// TIA Portal V19 export
FUNCTION_BLOCK "A02_HMI_FB"   // FB175, LAD
TITLE = HMI Managment
AUTHOR : Piemme
FAMILY : System
// stored: MemoryReserve 100, SetENOAutomatically false
   VAR
      MB2_Decoder { ExternalAccessible := 'False'; ExternalVisible := 'False'; ExternalWritable := 'False'} : "ButtonsHMIDecoder";
   END_VAR
   VAR_TEMP
      i : Int;
      tempIdxMove : Int;
      tempIdxPos : Int;
      tempIdxVert : Int;
      tempIdxHoriz : Int;
   END_VAR
   VAR CONSTANT
      "2001_HU_AREA02" : Int := 2001;
      "2011_PIT_TABLE1" : Int := 2011;
      "2021_ROLLFORMER_MOVE" : Int := 2021;
      "2022_ROLLFORMER_LUBR_1" : Int := 2022;
      "2023_ROLLFORMER_LUBR_2" : Int := 2023;
      "2024_ROLLFORMER_LUBR_3" : Int := 2024;
      "2031_MWFAKCALC_PUSHAX" : Int := 2031;
      "2032_MWFAKCALC_GRIPPER" : Int := 2032;
      "2041_FLYINGCARRIAGE_MOVE" : Int := 2041;
      "2042_FLYINGCARRIAGE_POS" : Int := 2042;
      "2043_FLYINGCARRIAGE_ZERO" : Int := 2043;
      "2044_FLYINGCARRIAGE_LUBR" : Int := 2044;
      "2051_FINALCUT_LOCKING" : Int := 2051;
      "2052_FINALCUT_CUTHEAD" : Int := 2052;
      "2053_FINALCUT_DRAWHEAD" : Int := 2053;
      "2054_FINALCUT_MARKHEAD" : Int := 2054;
      "2055_FINALCUT_LUBR" : Int := 2055;
      "2061_ACCROLLCONVEYOR_COMBO_MOVE" : Int := 2061;
      "2062_ACCROLLCONVEYOR_PUSHER_COMBO_VERT" : Int := 2062;
      "2063_ACCROLLCONVEYOR_PUSHER_COMBO_HORIZ" : Int := 2063;
      "2071_ACCROLLCONVEYOR_ROLL1" : Int := 2071;
      "2072_ACCROLLCONVEYOR_ROLL2" : Int := 2072;
      "2073_ACCROLLCONVEYOR_ROLL3" : Int := 2073;
      "2081_ACCROLLCONVEYOR_PUSHER_VERT_1" : Int := 2081;
      "2082_ACCROLLCONVEYOR_PUSHER_VERT_2" : Int := 2082;
      "2083_ACCROLLCONVEYOR_PUSHER_VERT_3" : Int := 2083;
      "2084_ACCROLLCONVEYOR_PUSHER_VERT_4" : Int := 2084;
      "2085_ACCROLLCONVEYOR_PUSHER_VERT_5" : Int := 2085;
      "2086_ACCROLLCONVEYOR_PUSHER_VERT_6" : Int := 2086;
      "2091_ACCROLLCONVEYOR_PUSHER_HORIZ_1" : Int := 2091;
      "2092_ACCROLLCONVEYOR_PUSHER_HORIZ_2" : Int := 2092;
      "2093_ACCROLLCONVEYOR_PUSHER_HORIZ_3" : Int := 2093;
      "2094_ACCROLLCONVEYOR_PUSHER_HORIZ_4" : Int := 2094;
      "2095_ACCROLLCONVEYOR_PUSHER_HORIZ_5" : Int := 2095;
      "2096_ACCROLLCONVEYOR_PUSHER_HORIZ_6" : Int := 2096;
      "2100_MODULO1_OP_MOVE" : Int := 2100;
      "2101_MODULO1_OP_POS" : Int := 2101;
      "2102_MODULO1_MOT_MOVE" : Int := 2102;
      "2103_MODULO1_MOT_POS" : Int := 2103;
      "2104_MODULO2_OP_MOVE" : Int := 2104;
      "2105_MODULO2_OP_POS" : Int := 2105;
      "2106_MODULO2_MOT_MOVE" : Int := 2106;
      "2107_MODULO2_MOT_POS" : Int := 2107;
      "2108_MODULO3_OP_MOVE" : Int := 2108;
      "2109_MODULO3_OP_POS" : Int := 2109;
      "2110_MODULO3_MOT_MOVE" : Int := 2110;
      "2111_MODULO3_MOT_POS" : Int := 2111;
      "2112_PASSAGGIO2_OP_MOVE" : Int := 2112;
      "2113_PASSAGGIO2_OP_POS" : Int := 2113;
      "2114_PASSAGGIO2_MOT_MOVE" : Int := 2114;
      "2115_PASSAGGIO2_MOT_POS" : Int := 2115;
      "2116_PASSAGGIO14_OP_MOVE" : Int := 2116;
      "2117_PASSAGGIO14_OP_POS" : Int := 2117;
      "2118_PASSAGGIO14_MOT_MOVE" : Int := 2118;
      "2119_PASSAGGIO14_MOT_POS" : Int := 2119;
      "2120_PASSAGGIO17_OP_MOVE" : Int := 2120;
      "2121_PASSAGGIO17_OP_POS" : Int := 2121;
      "2122_PASSAGGIO17_MOT_MOVE" : Int := 2122;
      "2123_PASSAGGIO17_MOT_POS" : Int := 2123;
      "2124_PASSAGGIO18_OP_MOVE" : Int := 2124;
      "2125_PASSAGGIO18_OP_POS" : Int := 2125;
      "2126_PASSAGGIO18_MOT_MOVE" : Int := 2126;
      "2127_PASSAGGIO18_MOT_POS" : Int := 2127;
      "2280_PASSAGGIO2_COMBO_MOVE" : Int := 2280;
      "2281_PASSAGGIO2_COMBO_POS" : Int := 2281;
      "2282_PASSAGGIO14_COMBO_MOVE" : Int := 2282;
      "2283_PASSAGGIO14_COMBO_POS" : Int := 2283;
      "2284_PASSAGGIO17_COMBO_MOVE" : Int := 2284;
      "2285_PASSAGGIO17_COMBO_POS" : Int := 2285;
      "2286_PASSAGGIO18_COMBO_MOVE" : Int := 2286;
      "2287_PASSAGGIO18_COMBO_POS" : Int := 2287;
   END_VAR
   VAR_TEMP   // added for the SCL form of the ladder/FBD networks
      _w1 : Bool;
   END_VAR
BEGIN

REGION Network 2: <<< MB2 MANUALS OPERATIONS >>>
END_REGION

REGION Network 3 (SCL): Reset Op
   #MB2_Decoder.OpEnabled := FALSE;
   #MB2_Decoder.OpRunning := FALSE;
   #MB2_Decoder.OpDone := FALSE;
END_REGION

REGION Network 4: MB2 Code 2001 - Area 02 HU
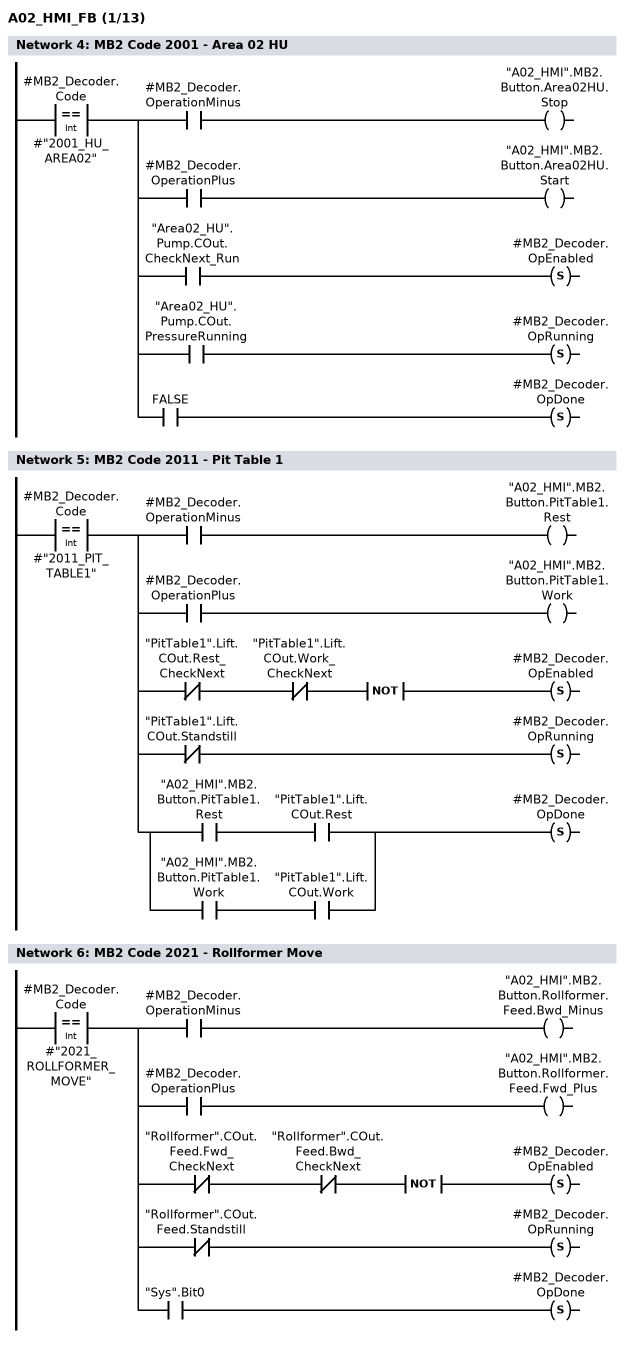
   RUNG wire#powerrail
      { S7_Templates := "SrcType := Int" } EQ_Contact(in1 := #MB2_Decoder.Code, in2 := #"2001_HU_AREA02")
      wire#w1
      Contact( #MB2_Decoder.OperationMinus )
      Coil( "A02_HMI".MB2.Button.Area02HU.Stop )
   END_RUNG
   RUNG wire#w1
      Contact( #MB2_Decoder.OperationPlus )
      Coil( "A02_HMI".MB2.Button.Area02HU.Start )
   END_RUNG
   RUNG wire#w1
      Contact( "Area02_HU".Pump.COut.CheckNext_Run )
      S_Coil( #MB2_Decoder.OpEnabled )
   END_RUNG
   RUNG wire#w1
      Contact( "Area02_HU".Pump.COut.PressureRunning )
      S_Coil( #MB2_Decoder.OpRunning )
   END_RUNG
   RUNG wire#w1
      Contact( FALSE )
      S_Coil( #MB2_Decoder.OpDone )
   END_RUNG
   // the same network as SCL:
   #_w1 := #MB2_Decoder.Code = #"2001_HU_AREA02";
   "A02_HMI".MB2.Button.Area02HU.Stop := #_w1 AND #MB2_Decoder.OperationMinus;
   "A02_HMI".MB2.Button.Area02HU.Start := #_w1 AND #MB2_Decoder.OperationPlus;
   IF #_w1 AND "Area02_HU".Pump.COut.CheckNext_Run THEN #MB2_Decoder.OpEnabled := TRUE; END_IF;
   IF #_w1 AND "Area02_HU".Pump.COut.PressureRunning THEN #MB2_Decoder.OpRunning := TRUE; END_IF;
   IF #_w1 AND FALSE THEN #MB2_Decoder.OpDone := TRUE; END_IF;
END_REGION

REGION Network 5: MB2 Code 2011 - Pit Table 1
   RUNG wire#powerrail
      { S7_Templates := "SrcType := Int" } EQ_Contact(in1 := #MB2_Decoder.Code, in2 := #"2011_PIT_TABLE1")
      wire#w1
      Contact( #MB2_Decoder.OperationMinus )
      Coil( "A02_HMI".MB2.Button.PitTable1.Rest )
   END_RUNG
   RUNG wire#w1
      Contact( #MB2_Decoder.OperationPlus )
      Coil( "A02_HMI".MB2.Button.PitTable1.Work )
   END_RUNG
   RUNG wire#w1
      I_Contact( "PitTable1".Lift.COut.Rest_CheckNext )
      I_Contact( "PitTable1".Lift.COut.Work_CheckNext )
      Not()
      S_Coil( #MB2_Decoder.OpEnabled )
   END_RUNG
   RUNG wire#w1
      I_Contact( "PitTable1".Lift.COut.Standstill )
      S_Coil( #MB2_Decoder.OpRunning )
   END_RUNG
   RUNG wire#w1
      Contact( "A02_HMI".MB2.Button.PitTable1.Rest )
      Contact( "PitTable1".Lift.COut.Rest )
      wire#w2
      S_Coil( #MB2_Decoder.OpDone )
   END_RUNG
   RUNG wire#w1
      Contact( "A02_HMI".MB2.Button.PitTable1.Work )
      Contact( "PitTable1".Lift.COut.Work )
   END_RUNG wire#w2
   // the same network as SCL:
   #_w1 := #MB2_Decoder.Code = #"2011_PIT_TABLE1";
   "A02_HMI".MB2.Button.PitTable1.Rest := #_w1 AND #MB2_Decoder.OperationMinus;
   "A02_HMI".MB2.Button.PitTable1.Work := #_w1 AND #MB2_Decoder.OperationPlus;
   IF NOT (#_w1 AND NOT "PitTable1".Lift.COut.Rest_CheckNext AND NOT "PitTable1".Lift.COut.Work_CheckNext) THEN
       #MB2_Decoder.OpEnabled := TRUE;
   END_IF;
   IF #_w1 AND NOT "PitTable1".Lift.COut.Standstill THEN #MB2_Decoder.OpRunning := TRUE; END_IF;
   IF #_w1 AND (("A02_HMI".MB2.Button.PitTable1.Rest AND "PitTable1".Lift.COut.Rest) OR ("A02_HMI".MB2.Button.PitTable1.Work AND "PitTable1".Lift.COut.Work)) THEN
       #MB2_Decoder.OpDone := TRUE;
   END_IF;
END_REGION

REGION Network 6: MB2 Code 2021 - Rollformer Move
   RUNG wire#powerrail
      { S7_Templates := "SrcType := Int" } EQ_Contact(in1 := #MB2_Decoder.Code, in2 := #"2021_ROLLFORMER_MOVE")
      wire#w1
      Contact( #MB2_Decoder.OperationMinus )
      Coil( "A02_HMI".MB2.Button.Rollformer.Feed.Bwd_Minus )
   END_RUNG
   RUNG wire#w1
      Contact( #MB2_Decoder.OperationPlus )
      Coil( "A02_HMI".MB2.Button.Rollformer.Feed.Fwd_Plus )
   END_RUNG
   RUNG wire#w1
      I_Contact( "Rollformer".COut.Feed.Fwd_CheckNext )
      I_Contact( "Rollformer".COut.Feed.Bwd_CheckNext )
      Not()
      S_Coil( #MB2_Decoder.OpEnabled )
   END_RUNG
   RUNG wire#w1
      I_Contact( "Rollformer".COut.Feed.Standstill )
      S_Coil( #MB2_Decoder.OpRunning )
   END_RUNG
   RUNG wire#w1
      Contact( "Sys".Bit0 )
      S_Coil( #MB2_Decoder.OpDone )
   END_RUNG
   // the same network as SCL:
   #_w1 := #MB2_Decoder.Code = #"2021_ROLLFORMER_MOVE";
   "A02_HMI".MB2.Button.Rollformer.Feed.Bwd_Minus := #_w1 AND #MB2_Decoder.OperationMinus;
   "A02_HMI".MB2.Button.Rollformer.Feed.Fwd_Plus := #_w1 AND #MB2_Decoder.OperationPlus;
   IF NOT (#_w1 AND NOT "Rollformer".COut.Feed.Fwd_CheckNext AND NOT "Rollformer".COut.Feed.Bwd_CheckNext) THEN
       #MB2_Decoder.OpEnabled := TRUE;
   END_IF;
   IF #_w1 AND NOT "Rollformer".COut.Feed.Standstill THEN #MB2_Decoder.OpRunning := TRUE; END_IF;
   IF #_w1 AND "Sys".Bit0 THEN #MB2_Decoder.OpDone := TRUE; END_IF;
END_REGION

REGION Network 7: MB2 Code 2022 - Rollformer Lubr 1
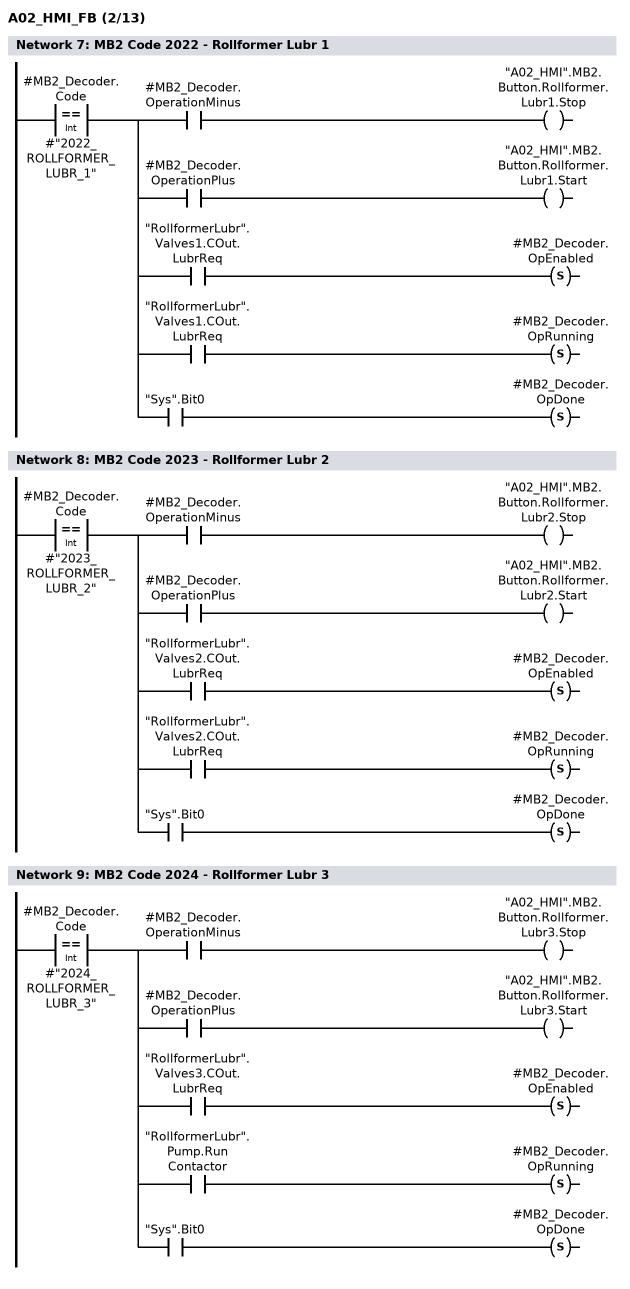
   RUNG wire#powerrail
      { S7_Templates := "SrcType := Int" } EQ_Contact(in1 := #MB2_Decoder.Code, in2 := #"2022_ROLLFORMER_LUBR_1")
      wire#w1
      Contact( #MB2_Decoder.OperationMinus )
      Coil( "A02_HMI".MB2.Button.Rollformer.Lubr1.Stop )
   END_RUNG
   RUNG wire#w1
      Contact( #MB2_Decoder.OperationPlus )
      Coil( "A02_HMI".MB2.Button.Rollformer.Lubr1.Start )
   END_RUNG
   RUNG wire#w1
      Contact( "RollformerLubr".Valves1.COut.LubrReq )
      S_Coil( #MB2_Decoder.OpEnabled )
   END_RUNG
   RUNG wire#w1
      Contact( "RollformerLubr".Valves1.COut.LubrReq )
      S_Coil( #MB2_Decoder.OpRunning )
   END_RUNG
   RUNG wire#w1
      Contact( "Sys".Bit0 )
      S_Coil( #MB2_Decoder.OpDone )
   END_RUNG
   // the same network as SCL:
   #_w1 := #MB2_Decoder.Code = #"2022_ROLLFORMER_LUBR_1";
   "A02_HMI".MB2.Button.Rollformer.Lubr1.Stop := #_w1 AND #MB2_Decoder.OperationMinus;
   "A02_HMI".MB2.Button.Rollformer.Lubr1.Start := #_w1 AND #MB2_Decoder.OperationPlus;
   IF #_w1 AND "RollformerLubr".Valves1.COut.LubrReq THEN
       #MB2_Decoder.OpEnabled := TRUE;
       #MB2_Decoder.OpRunning := TRUE;
   END_IF;
   IF #_w1 AND "Sys".Bit0 THEN #MB2_Decoder.OpDone := TRUE; END_IF;
END_REGION

REGION Network 8: MB2 Code 2023 - Rollformer Lubr 2
   RUNG wire#powerrail
      { S7_Templates := "SrcType := Int" } EQ_Contact(in1 := #MB2_Decoder.Code, in2 := #"2023_ROLLFORMER_LUBR_2")
      wire#w1
      Contact( #MB2_Decoder.OperationMinus )
      Coil( "A02_HMI".MB2.Button.Rollformer.Lubr2.Stop )
   END_RUNG
   RUNG wire#w1
      Contact( #MB2_Decoder.OperationPlus )
      Coil( "A02_HMI".MB2.Button.Rollformer.Lubr2.Start )
   END_RUNG
   RUNG wire#w1
      Contact( "RollformerLubr".Valves2.COut.LubrReq )
      S_Coil( #MB2_Decoder.OpEnabled )
   END_RUNG
   RUNG wire#w1
      Contact( "RollformerLubr".Valves2.COut.LubrReq )
      S_Coil( #MB2_Decoder.OpRunning )
   END_RUNG
   RUNG wire#w1
      Contact( "Sys".Bit0 )
      S_Coil( #MB2_Decoder.OpDone )
   END_RUNG
   // the same network as SCL:
   #_w1 := #MB2_Decoder.Code = #"2023_ROLLFORMER_LUBR_2";
   "A02_HMI".MB2.Button.Rollformer.Lubr2.Stop := #_w1 AND #MB2_Decoder.OperationMinus;
   "A02_HMI".MB2.Button.Rollformer.Lubr2.Start := #_w1 AND #MB2_Decoder.OperationPlus;
   IF #_w1 AND "RollformerLubr".Valves2.COut.LubrReq THEN
       #MB2_Decoder.OpEnabled := TRUE;
       #MB2_Decoder.OpRunning := TRUE;
   END_IF;
   IF #_w1 AND "Sys".Bit0 THEN #MB2_Decoder.OpDone := TRUE; END_IF;
END_REGION

REGION Network 9: MB2 Code 2024 - Rollformer Lubr 3
   RUNG wire#powerrail
      { S7_Templates := "SrcType := Int" } EQ_Contact(in1 := #MB2_Decoder.Code, in2 := #"2024_ROLLFORMER_LUBR_3")
      wire#w1
      Contact( #MB2_Decoder.OperationMinus )
      Coil( "A02_HMI".MB2.Button.Rollformer.Lubr3.Stop )
   END_RUNG
   RUNG wire#w1
      Contact( #MB2_Decoder.OperationPlus )
      Coil( "A02_HMI".MB2.Button.Rollformer.Lubr3.Start )
   END_RUNG
   RUNG wire#w1
      Contact( "RollformerLubr".Valves3.COut.LubrReq )
      S_Coil( #MB2_Decoder.OpEnabled )
   END_RUNG
   RUNG wire#w1
      Contact( "RollformerLubr".Pump.RunContactor )
      S_Coil( #MB2_Decoder.OpRunning )
   END_RUNG
   RUNG wire#w1
      Contact( "Sys".Bit0 )
      S_Coil( #MB2_Decoder.OpDone )
   END_RUNG
   // the same network as SCL:
   #_w1 := #MB2_Decoder.Code = #"2024_ROLLFORMER_LUBR_3";
   "A02_HMI".MB2.Button.Rollformer.Lubr3.Stop := #_w1 AND #MB2_Decoder.OperationMinus;
   "A02_HMI".MB2.Button.Rollformer.Lubr3.Start := #_w1 AND #MB2_Decoder.OperationPlus;
   IF #_w1 AND "RollformerLubr".Valves3.COut.LubrReq THEN #MB2_Decoder.OpEnabled := TRUE; END_IF;
   IF #_w1 AND "RollformerLubr".Pump.RunContactor THEN #MB2_Decoder.OpRunning := TRUE; END_IF;
   IF #_w1 AND "Sys".Bit0 THEN #MB2_Decoder.OpDone := TRUE; END_IF;
END_REGION

REGION Network 10: MB2 Code 2031 - MwFakCalc push ax
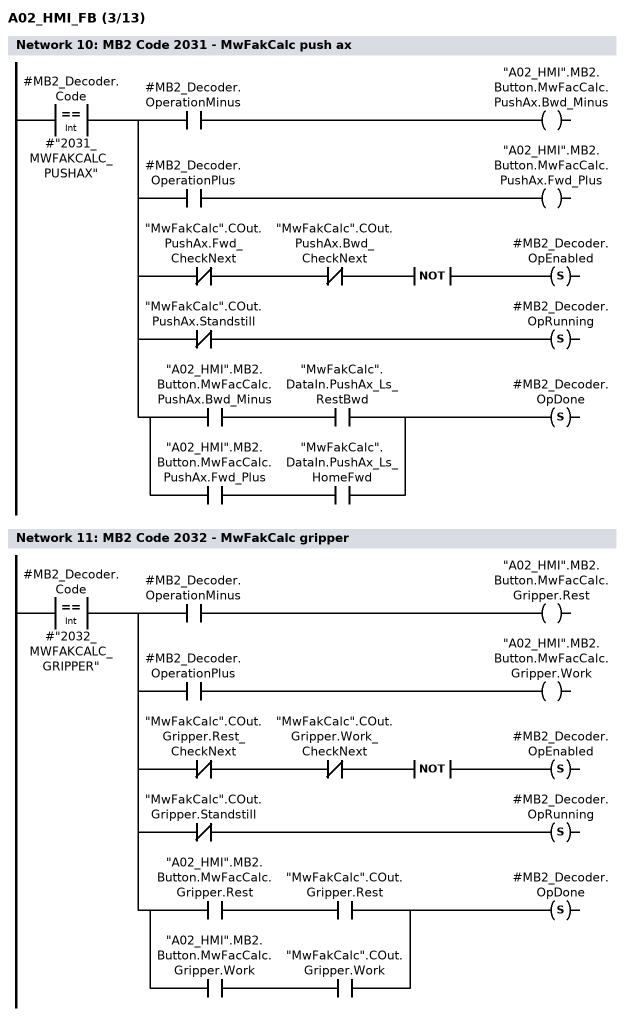
   RUNG wire#powerrail
      { S7_Templates := "SrcType := Int" } EQ_Contact(in1 := #MB2_Decoder.Code, in2 := #"2031_MWFAKCALC_PUSHAX")
      wire#w1
      Contact( #MB2_Decoder.OperationMinus )
      Coil( "A02_HMI".MB2.Button.MwFacCalc.PushAx.Bwd_Minus )
   END_RUNG
   RUNG wire#w1
      Contact( #MB2_Decoder.OperationPlus )
      Coil( "A02_HMI".MB2.Button.MwFacCalc.PushAx.Fwd_Plus )
   END_RUNG
   RUNG wire#w1
      I_Contact( "MwFakCalc".COut.PushAx.Fwd_CheckNext )
      I_Contact( "MwFakCalc".COut.PushAx.Bwd_CheckNext )
      Not()
      S_Coil( #MB2_Decoder.OpEnabled )
   END_RUNG
   RUNG wire#w1
      I_Contact( "MwFakCalc".COut.PushAx.Standstill )
      S_Coil( #MB2_Decoder.OpRunning )
   END_RUNG
   RUNG wire#w1
      Contact( "A02_HMI".MB2.Button.MwFacCalc.PushAx.Bwd_Minus )
      Contact( "MwFakCalc".DataIn.PushAx_Ls_RestBwd )
      wire#w2
      S_Coil( #MB2_Decoder.OpDone )
   END_RUNG
   RUNG wire#w1
      Contact( "A02_HMI".MB2.Button.MwFacCalc.PushAx.Fwd_Plus )
      Contact( "MwFakCalc".DataIn.PushAx_Ls_HomeFwd )
   END_RUNG wire#w2
   // the same network as SCL:
   #_w1 := #MB2_Decoder.Code = #"2031_MWFAKCALC_PUSHAX";
   "A02_HMI".MB2.Button.MwFacCalc.PushAx.Bwd_Minus := #_w1 AND #MB2_Decoder.OperationMinus;
   "A02_HMI".MB2.Button.MwFacCalc.PushAx.Fwd_Plus := #_w1 AND #MB2_Decoder.OperationPlus;
   IF NOT (#_w1 AND NOT "MwFakCalc".COut.PushAx.Fwd_CheckNext AND NOT "MwFakCalc".COut.PushAx.Bwd_CheckNext) THEN
       #MB2_Decoder.OpEnabled := TRUE;
   END_IF;
   IF #_w1 AND NOT "MwFakCalc".COut.PushAx.Standstill THEN #MB2_Decoder.OpRunning := TRUE; END_IF;
   IF #_w1 AND (("A02_HMI".MB2.Button.MwFacCalc.PushAx.Bwd_Minus AND "MwFakCalc".DataIn.PushAx_Ls_RestBwd) OR ("A02_HMI".MB2.Button.MwFacCalc.PushAx.Fwd_Plus AND "MwFakCalc".DataIn.PushAx_Ls_HomeFwd)) THEN
       #MB2_Decoder.OpDone := TRUE;
   END_IF;
END_REGION

REGION Network 11: MB2 Code 2032 - MwFakCalc gripper
   RUNG wire#powerrail
      { S7_Templates := "SrcType := Int" } EQ_Contact(in1 := #MB2_Decoder.Code, in2 := #"2032_MWFAKCALC_GRIPPER")
      wire#w1
      Contact( #MB2_Decoder.OperationMinus )
      Coil( "A02_HMI".MB2.Button.MwFacCalc.Gripper.Rest )
   END_RUNG
   RUNG wire#w1
      Contact( #MB2_Decoder.OperationPlus )
      Coil( "A02_HMI".MB2.Button.MwFacCalc.Gripper.Work )
   END_RUNG
   RUNG wire#w1
      I_Contact( "MwFakCalc".COut.Gripper.Rest_CheckNext )
      I_Contact( "MwFakCalc".COut.Gripper.Work_CheckNext )
      Not()
      S_Coil( #MB2_Decoder.OpEnabled )
   END_RUNG
   RUNG wire#w1
      I_Contact( "MwFakCalc".COut.Gripper.Standstill )
      S_Coil( #MB2_Decoder.OpRunning )
   END_RUNG
   RUNG wire#w1
      Contact( "A02_HMI".MB2.Button.MwFacCalc.Gripper.Rest )
      Contact( "MwFakCalc".COut.Gripper.Rest )
      wire#w2
      S_Coil( #MB2_Decoder.OpDone )
   END_RUNG
   RUNG wire#w1
      Contact( "A02_HMI".MB2.Button.MwFacCalc.Gripper.Work )
      Contact( "MwFakCalc".COut.Gripper.Work )
   END_RUNG wire#w2
   // the same network as SCL:
   #_w1 := #MB2_Decoder.Code = #"2032_MWFAKCALC_GRIPPER";
   "A02_HMI".MB2.Button.MwFacCalc.Gripper.Rest := #_w1 AND #MB2_Decoder.OperationMinus;
   "A02_HMI".MB2.Button.MwFacCalc.Gripper.Work := #_w1 AND #MB2_Decoder.OperationPlus;
   IF NOT (#_w1 AND NOT "MwFakCalc".COut.Gripper.Rest_CheckNext AND NOT "MwFakCalc".COut.Gripper.Work_CheckNext) THEN
       #MB2_Decoder.OpEnabled := TRUE;
   END_IF;
   IF #_w1 AND NOT "MwFakCalc".COut.Gripper.Standstill THEN #MB2_Decoder.OpRunning := TRUE; END_IF;
   IF #_w1 AND (("A02_HMI".MB2.Button.MwFacCalc.Gripper.Rest AND "MwFakCalc".COut.Gripper.Rest) OR ("A02_HMI".MB2.Button.MwFacCalc.Gripper.Work AND "MwFakCalc".COut.Gripper.Work)) THEN
       #MB2_Decoder.OpDone := TRUE;
   END_IF;
END_REGION

REGION Network 12: MB2 Code 2041 - Flying carriage move
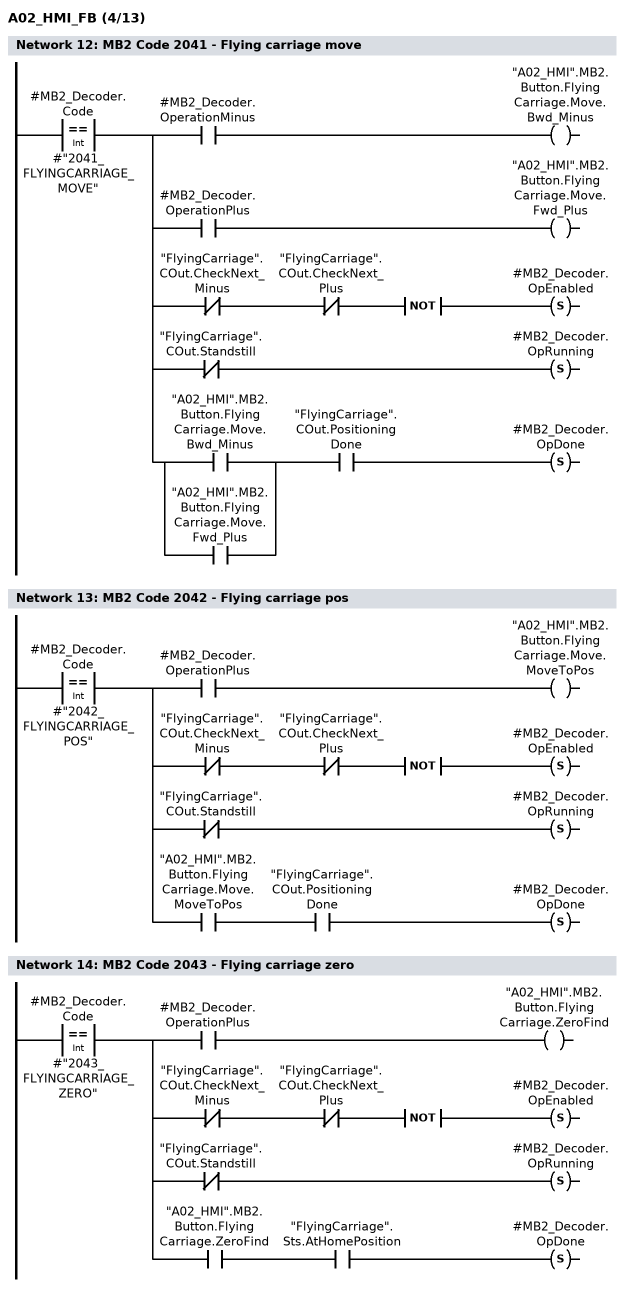
   RUNG wire#powerrail
      { S7_Templates := "SrcType := Int" } EQ_Contact(in1 := #MB2_Decoder.Code, in2 := #"2041_FLYINGCARRIAGE_MOVE")
      wire#w1
      Contact( #MB2_Decoder.OperationMinus )
      Coil( "A02_HMI".MB2.Button.FlyingCarriage.Move.Bwd_Minus )
   END_RUNG
   RUNG wire#w1
      Contact( #MB2_Decoder.OperationPlus )
      Coil( "A02_HMI".MB2.Button.FlyingCarriage.Move.Fwd_Plus )
   END_RUNG
   RUNG wire#w1
      I_Contact( "FlyingCarriage".COut.CheckNext_Minus )
      I_Contact( "FlyingCarriage".COut.CheckNext_Plus )
      Not()
      S_Coil( #MB2_Decoder.OpEnabled )
   END_RUNG
   RUNG wire#w1
      I_Contact( "FlyingCarriage".COut.Standstill )
      S_Coil( #MB2_Decoder.OpRunning )
   END_RUNG
   RUNG wire#w1
      Contact( "A02_HMI".MB2.Button.FlyingCarriage.Move.Bwd_Minus )
      wire#w2
      Contact( "FlyingCarriage".COut.PositioningDone )
      S_Coil( #MB2_Decoder.OpDone )
   END_RUNG
   RUNG wire#w1
      Contact( "A02_HMI".MB2.Button.FlyingCarriage.Move.Fwd_Plus )
   END_RUNG wire#w2
   // the same network as SCL:
   #_w1 := #MB2_Decoder.Code = #"2041_FLYINGCARRIAGE_MOVE";
   "A02_HMI".MB2.Button.FlyingCarriage.Move.Bwd_Minus := #_w1 AND #MB2_Decoder.OperationMinus;
   "A02_HMI".MB2.Button.FlyingCarriage.Move.Fwd_Plus := #_w1 AND #MB2_Decoder.OperationPlus;
   IF NOT (#_w1 AND NOT "FlyingCarriage".COut.CheckNext_Minus AND NOT "FlyingCarriage".COut.CheckNext_Plus) THEN
       #MB2_Decoder.OpEnabled := TRUE;
   END_IF;
   IF #_w1 AND NOT "FlyingCarriage".COut.Standstill THEN #MB2_Decoder.OpRunning := TRUE; END_IF;
   IF #_w1 AND ("A02_HMI".MB2.Button.FlyingCarriage.Move.Bwd_Minus OR "A02_HMI".MB2.Button.FlyingCarriage.Move.Fwd_Plus) AND "FlyingCarriage".COut.PositioningDone THEN
       #MB2_Decoder.OpDone := TRUE;
   END_IF;
END_REGION

REGION Network 13: MB2 Code 2042 - Flying carriage pos
   RUNG wire#powerrail
      { S7_Templates := "SrcType := Int" } EQ_Contact(in1 := #MB2_Decoder.Code, in2 := #"2042_FLYINGCARRIAGE_POS")
      wire#w1
      Contact( #MB2_Decoder.OperationPlus )
      Coil( "A02_HMI".MB2.Button.FlyingCarriage.Move.MoveToPos )
   END_RUNG
   RUNG wire#w1
      I_Contact( "FlyingCarriage".COut.CheckNext_Minus )
      I_Contact( "FlyingCarriage".COut.CheckNext_Plus )
      Not()
      S_Coil( #MB2_Decoder.OpEnabled )
   END_RUNG
   RUNG wire#w1
      I_Contact( "FlyingCarriage".COut.Standstill )
      S_Coil( #MB2_Decoder.OpRunning )
   END_RUNG
   RUNG wire#w1
      Contact( "A02_HMI".MB2.Button.FlyingCarriage.Move.MoveToPos )
      Contact( "FlyingCarriage".COut.PositioningDone )
      S_Coil( #MB2_Decoder.OpDone )
   END_RUNG
   // the same network as SCL:
   #_w1 := #MB2_Decoder.Code = #"2042_FLYINGCARRIAGE_POS";
   "A02_HMI".MB2.Button.FlyingCarriage.Move.MoveToPos := #_w1 AND #MB2_Decoder.OperationPlus;
   IF NOT (#_w1 AND NOT "FlyingCarriage".COut.CheckNext_Minus AND NOT "FlyingCarriage".COut.CheckNext_Plus) THEN
       #MB2_Decoder.OpEnabled := TRUE;
   END_IF;
   IF #_w1 AND NOT "FlyingCarriage".COut.Standstill THEN #MB2_Decoder.OpRunning := TRUE; END_IF;
   IF #_w1 AND "A02_HMI".MB2.Button.FlyingCarriage.Move.MoveToPos AND "FlyingCarriage".COut.PositioningDone THEN
       #MB2_Decoder.OpDone := TRUE;
   END_IF;
END_REGION

REGION Network 14: MB2 Code 2043 - Flying carriage zero
   RUNG wire#powerrail
      { S7_Templates := "SrcType := Int" } EQ_Contact(in1 := #MB2_Decoder.Code, in2 := #"2043_FLYINGCARRIAGE_ZERO")
      wire#w1
      Contact( #MB2_Decoder.OperationPlus )
      Coil( "A02_HMI".MB2.Button.FlyingCarriage.ZeroFind )
   END_RUNG
   RUNG wire#w1
      I_Contact( "FlyingCarriage".COut.CheckNext_Minus )
      I_Contact( "FlyingCarriage".COut.CheckNext_Plus )
      Not()
      S_Coil( #MB2_Decoder.OpEnabled )
   END_RUNG
   RUNG wire#w1
      I_Contact( "FlyingCarriage".COut.Standstill )
      S_Coil( #MB2_Decoder.OpRunning )
   END_RUNG
   RUNG wire#w1
      Contact( "A02_HMI".MB2.Button.FlyingCarriage.ZeroFind )
      Contact( "FlyingCarriage".Sts.AtHomePosition )
      S_Coil( #MB2_Decoder.OpDone )
   END_RUNG
   // the same network as SCL:
   #_w1 := #MB2_Decoder.Code = #"2043_FLYINGCARRIAGE_ZERO";
   "A02_HMI".MB2.Button.FlyingCarriage.ZeroFind := #_w1 AND #MB2_Decoder.OperationPlus;
   IF NOT (#_w1 AND NOT "FlyingCarriage".COut.CheckNext_Minus AND NOT "FlyingCarriage".COut.CheckNext_Plus) THEN
       #MB2_Decoder.OpEnabled := TRUE;
   END_IF;
   IF #_w1 AND NOT "FlyingCarriage".COut.Standstill THEN #MB2_Decoder.OpRunning := TRUE; END_IF;
   IF #_w1 AND "A02_HMI".MB2.Button.FlyingCarriage.ZeroFind AND "FlyingCarriage".Sts.AtHomePosition THEN
       #MB2_Decoder.OpDone := TRUE;
   END_IF;
END_REGION

REGION Network 15: MB2 Code 2044 - Flying carriage lubr
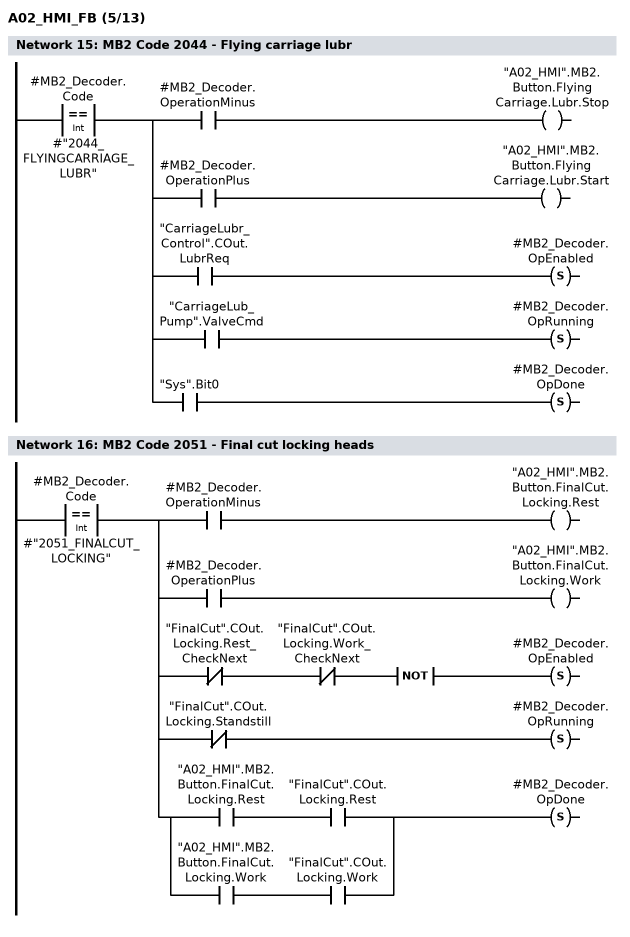
   RUNG wire#powerrail
      { S7_Templates := "SrcType := Int" } EQ_Contact(in1 := #MB2_Decoder.Code, in2 := #"2044_FLYINGCARRIAGE_LUBR")
      wire#w1
      Contact( #MB2_Decoder.OperationMinus )
      Coil( "A02_HMI".MB2.Button.FlyingCarriage.Lubr.Stop )
   END_RUNG
   RUNG wire#w1
      Contact( #MB2_Decoder.OperationPlus )
      Coil( "A02_HMI".MB2.Button.FlyingCarriage.Lubr.Start )
   END_RUNG
   RUNG wire#w1
      Contact( "CarriageLubr_Control".COut.LubrReq )
      S_Coil( #MB2_Decoder.OpEnabled )
   END_RUNG
   RUNG wire#w1
      Contact( "CarriageLub_Pump".ValveCmd )
      S_Coil( #MB2_Decoder.OpRunning )
   END_RUNG
   RUNG wire#w1
      Contact( "Sys".Bit0 )
      S_Coil( #MB2_Decoder.OpDone )
   END_RUNG
   // the same network as SCL:
   #_w1 := #MB2_Decoder.Code = #"2044_FLYINGCARRIAGE_LUBR";
   "A02_HMI".MB2.Button.FlyingCarriage.Lubr.Stop := #_w1 AND #MB2_Decoder.OperationMinus;
   "A02_HMI".MB2.Button.FlyingCarriage.Lubr.Start := #_w1 AND #MB2_Decoder.OperationPlus;
   IF #_w1 AND "CarriageLubr_Control".COut.LubrReq THEN #MB2_Decoder.OpEnabled := TRUE; END_IF;
   IF #_w1 AND "CarriageLub_Pump".ValveCmd THEN #MB2_Decoder.OpRunning := TRUE; END_IF;
   IF #_w1 AND "Sys".Bit0 THEN #MB2_Decoder.OpDone := TRUE; END_IF;
END_REGION

REGION Network 16: MB2 Code 2051 - Final cut locking heads
   RUNG wire#powerrail
      { S7_Templates := "SrcType := Int" } EQ_Contact(in1 := #MB2_Decoder.Code, in2 := #"2051_FINALCUT_LOCKING")
      wire#w1
      Contact( #MB2_Decoder.OperationMinus )
      Coil( "A02_HMI".MB2.Button.FinalCut.Locking.Rest )
   END_RUNG
   RUNG wire#w1
      Contact( #MB2_Decoder.OperationPlus )
      Coil( "A02_HMI".MB2.Button.FinalCut.Locking.Work )
   END_RUNG
   RUNG wire#w1
      I_Contact( "FinalCut".COut.Locking.Rest_CheckNext )
      I_Contact( "FinalCut".COut.Locking.Work_CheckNext )
      Not()
      S_Coil( #MB2_Decoder.OpEnabled )
   END_RUNG
   RUNG wire#w1
      I_Contact( "FinalCut".COut.Locking.Standstill )
      S_Coil( #MB2_Decoder.OpRunning )
   END_RUNG
   RUNG wire#w1
      Contact( "A02_HMI".MB2.Button.FinalCut.Locking.Rest )
      Contact( "FinalCut".COut.Locking.Rest )
      wire#w2
      S_Coil( #MB2_Decoder.OpDone )
   END_RUNG
   RUNG wire#w1
      Contact( "A02_HMI".MB2.Button.FinalCut.Locking.Work )
      Contact( "FinalCut".COut.Locking.Work )
   END_RUNG wire#w2
   // the same network as SCL:
   #_w1 := #MB2_Decoder.Code = #"2051_FINALCUT_LOCKING";
   "A02_HMI".MB2.Button.FinalCut.Locking.Rest := #_w1 AND #MB2_Decoder.OperationMinus;
   "A02_HMI".MB2.Button.FinalCut.Locking.Work := #_w1 AND #MB2_Decoder.OperationPlus;
   IF NOT (#_w1 AND NOT "FinalCut".COut.Locking.Rest_CheckNext AND NOT "FinalCut".COut.Locking.Work_CheckNext) THEN
       #MB2_Decoder.OpEnabled := TRUE;
   END_IF;
   IF #_w1 AND NOT "FinalCut".COut.Locking.Standstill THEN #MB2_Decoder.OpRunning := TRUE; END_IF;
   IF #_w1 AND (("A02_HMI".MB2.Button.FinalCut.Locking.Rest AND "FinalCut".COut.Locking.Rest) OR ("A02_HMI".MB2.Button.FinalCut.Locking.Work AND "FinalCut".COut.Locking.Work)) THEN
       #MB2_Decoder.OpDone := TRUE;
   END_IF;
END_REGION

REGION Network 17: MB2 Code 2052 - Final cut cut head
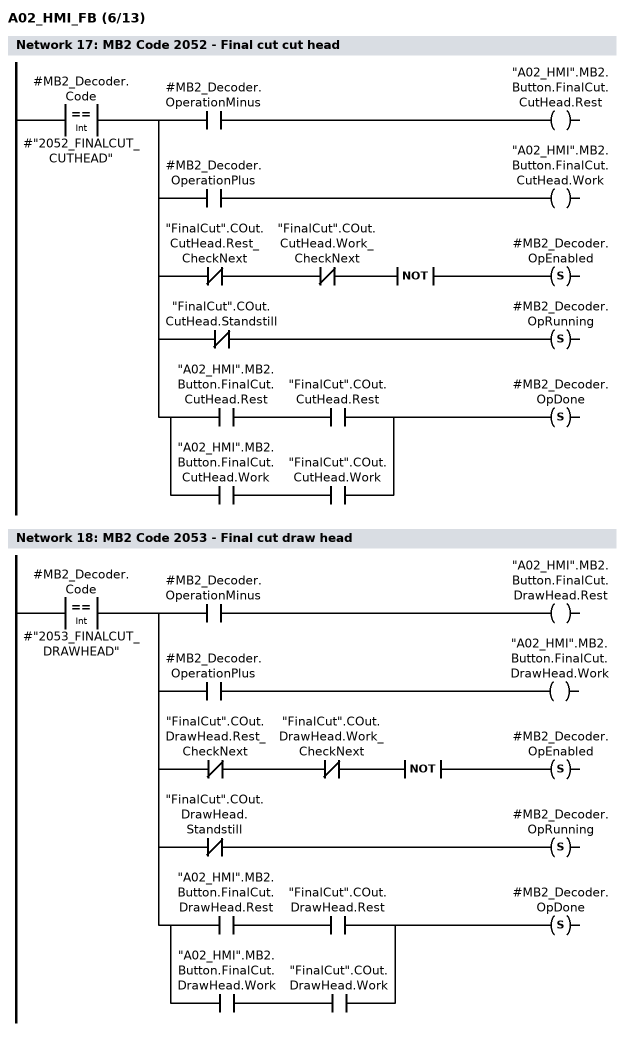
   RUNG wire#powerrail
      { S7_Templates := "SrcType := Int" } EQ_Contact(in1 := #MB2_Decoder.Code, in2 := #"2052_FINALCUT_CUTHEAD")
      wire#w1
      Contact( #MB2_Decoder.OperationMinus )
      Coil( "A02_HMI".MB2.Button.FinalCut.CutHead.Rest )
   END_RUNG
   RUNG wire#w1
      Contact( #MB2_Decoder.OperationPlus )
      Coil( "A02_HMI".MB2.Button.FinalCut.CutHead.Work )
   END_RUNG
   RUNG wire#w1
      I_Contact( "FinalCut".COut.CutHead.Rest_CheckNext )
      I_Contact( "FinalCut".COut.CutHead.Work_CheckNext )
      Not()
      S_Coil( #MB2_Decoder.OpEnabled )
   END_RUNG
   RUNG wire#w1
      I_Contact( "FinalCut".COut.CutHead.Standstill )
      S_Coil( #MB2_Decoder.OpRunning )
   END_RUNG
   RUNG wire#w1
      Contact( "A02_HMI".MB2.Button.FinalCut.CutHead.Rest )
      Contact( "FinalCut".COut.CutHead.Rest )
      wire#w2
      S_Coil( #MB2_Decoder.OpDone )
   END_RUNG
   RUNG wire#w1
      Contact( "A02_HMI".MB2.Button.FinalCut.CutHead.Work )
      Contact( "FinalCut".COut.CutHead.Work )
   END_RUNG wire#w2
   // the same network as SCL:
   #_w1 := #MB2_Decoder.Code = #"2052_FINALCUT_CUTHEAD";
   "A02_HMI".MB2.Button.FinalCut.CutHead.Rest := #_w1 AND #MB2_Decoder.OperationMinus;
   "A02_HMI".MB2.Button.FinalCut.CutHead.Work := #_w1 AND #MB2_Decoder.OperationPlus;
   IF NOT (#_w1 AND NOT "FinalCut".COut.CutHead.Rest_CheckNext AND NOT "FinalCut".COut.CutHead.Work_CheckNext) THEN
       #MB2_Decoder.OpEnabled := TRUE;
   END_IF;
   IF #_w1 AND NOT "FinalCut".COut.CutHead.Standstill THEN #MB2_Decoder.OpRunning := TRUE; END_IF;
   IF #_w1 AND (("A02_HMI".MB2.Button.FinalCut.CutHead.Rest AND "FinalCut".COut.CutHead.Rest) OR ("A02_HMI".MB2.Button.FinalCut.CutHead.Work AND "FinalCut".COut.CutHead.Work)) THEN
       #MB2_Decoder.OpDone := TRUE;
   END_IF;
END_REGION

REGION Network 18: MB2 Code 2053 - Final cut draw head
   RUNG wire#powerrail
      { S7_Templates := "SrcType := Int" } EQ_Contact(in1 := #MB2_Decoder.Code, in2 := #"2053_FINALCUT_DRAWHEAD")
      wire#w1
      Contact( #MB2_Decoder.OperationMinus )
      Coil( "A02_HMI".MB2.Button.FinalCut.DrawHead.Rest )
   END_RUNG
   RUNG wire#w1
      Contact( #MB2_Decoder.OperationPlus )
      Coil( "A02_HMI".MB2.Button.FinalCut.DrawHead.Work )
   END_RUNG
   RUNG wire#w1
      I_Contact( "FinalCut".COut.DrawHead.Rest_CheckNext )
      I_Contact( "FinalCut".COut.DrawHead.Work_CheckNext )
      Not()
      S_Coil( #MB2_Decoder.OpEnabled )
   END_RUNG
   RUNG wire#w1
      I_Contact( "FinalCut".COut.DrawHead.Standstill )
      S_Coil( #MB2_Decoder.OpRunning )
   END_RUNG
   RUNG wire#w1
      Contact( "A02_HMI".MB2.Button.FinalCut.DrawHead.Rest )
      Contact( "FinalCut".COut.DrawHead.Rest )
      wire#w2
      S_Coil( #MB2_Decoder.OpDone )
   END_RUNG
   RUNG wire#w1
      Contact( "A02_HMI".MB2.Button.FinalCut.DrawHead.Work )
      Contact( "FinalCut".COut.DrawHead.Work )
   END_RUNG wire#w2
   // the same network as SCL:
   #_w1 := #MB2_Decoder.Code = #"2053_FINALCUT_DRAWHEAD";
   "A02_HMI".MB2.Button.FinalCut.DrawHead.Rest := #_w1 AND #MB2_Decoder.OperationMinus;
   "A02_HMI".MB2.Button.FinalCut.DrawHead.Work := #_w1 AND #MB2_Decoder.OperationPlus;
   IF NOT (#_w1 AND NOT "FinalCut".COut.DrawHead.Rest_CheckNext AND NOT "FinalCut".COut.DrawHead.Work_CheckNext) THEN
       #MB2_Decoder.OpEnabled := TRUE;
   END_IF;
   IF #_w1 AND NOT "FinalCut".COut.DrawHead.Standstill THEN #MB2_Decoder.OpRunning := TRUE; END_IF;
   IF #_w1 AND (("A02_HMI".MB2.Button.FinalCut.DrawHead.Rest AND "FinalCut".COut.DrawHead.Rest) OR ("A02_HMI".MB2.Button.FinalCut.DrawHead.Work AND "FinalCut".COut.DrawHead.Work)) THEN
       #MB2_Decoder.OpDone := TRUE;
   END_IF;
END_REGION

REGION Network 19: MB2 Code 2054 - Final cut mark head
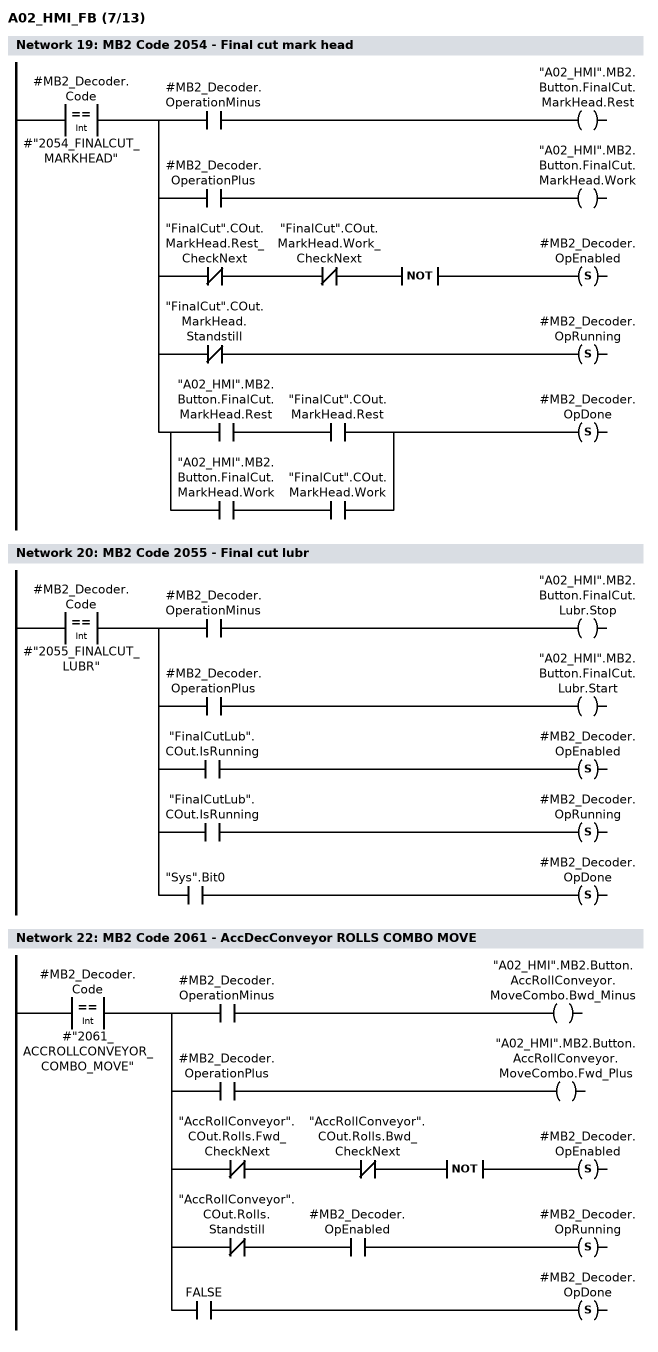
   RUNG wire#powerrail
      { S7_Templates := "SrcType := Int" } EQ_Contact(in1 := #MB2_Decoder.Code, in2 := #"2054_FINALCUT_MARKHEAD")
      wire#w1
      Contact( #MB2_Decoder.OperationMinus )
      Coil( "A02_HMI".MB2.Button.FinalCut.MarkHead.Rest )
   END_RUNG
   RUNG wire#w1
      Contact( #MB2_Decoder.OperationPlus )
      Coil( "A02_HMI".MB2.Button.FinalCut.MarkHead.Work )
   END_RUNG
   RUNG wire#w1
      I_Contact( "FinalCut".COut.MarkHead.Rest_CheckNext )
      I_Contact( "FinalCut".COut.MarkHead.Work_CheckNext )
      Not()
      S_Coil( #MB2_Decoder.OpEnabled )
   END_RUNG
   RUNG wire#w1
      I_Contact( "FinalCut".COut.MarkHead.Standstill )
      S_Coil( #MB2_Decoder.OpRunning )
   END_RUNG
   RUNG wire#w1
      Contact( "A02_HMI".MB2.Button.FinalCut.MarkHead.Rest )
      Contact( "FinalCut".COut.MarkHead.Rest )
      wire#w2
      S_Coil( #MB2_Decoder.OpDone )
   END_RUNG
   RUNG wire#w1
      Contact( "A02_HMI".MB2.Button.FinalCut.MarkHead.Work )
      Contact( "FinalCut".COut.MarkHead.Work )
   END_RUNG wire#w2
   // the same network as SCL:
   #_w1 := #MB2_Decoder.Code = #"2054_FINALCUT_MARKHEAD";
   "A02_HMI".MB2.Button.FinalCut.MarkHead.Rest := #_w1 AND #MB2_Decoder.OperationMinus;
   "A02_HMI".MB2.Button.FinalCut.MarkHead.Work := #_w1 AND #MB2_Decoder.OperationPlus;
   IF NOT (#_w1 AND NOT "FinalCut".COut.MarkHead.Rest_CheckNext AND NOT "FinalCut".COut.MarkHead.Work_CheckNext) THEN
       #MB2_Decoder.OpEnabled := TRUE;
   END_IF;
   IF #_w1 AND NOT "FinalCut".COut.MarkHead.Standstill THEN #MB2_Decoder.OpRunning := TRUE; END_IF;
   IF #_w1 AND (("A02_HMI".MB2.Button.FinalCut.MarkHead.Rest AND "FinalCut".COut.MarkHead.Rest) OR ("A02_HMI".MB2.Button.FinalCut.MarkHead.Work AND "FinalCut".COut.MarkHead.Work)) THEN
       #MB2_Decoder.OpDone := TRUE;
   END_IF;
END_REGION

REGION Network 20: MB2 Code 2055 - Final cut lubr
   RUNG wire#powerrail
      { S7_Templates := "SrcType := Int" } EQ_Contact(in1 := #MB2_Decoder.Code, in2 := #"2055_FINALCUT_LUBR")
      wire#w1
      Contact( #MB2_Decoder.OperationMinus )
      Coil( "A02_HMI".MB2.Button.FinalCut.Lubr.Stop )
   END_RUNG
   RUNG wire#w1
      Contact( #MB2_Decoder.OperationPlus )
      Coil( "A02_HMI".MB2.Button.FinalCut.Lubr.Start )
   END_RUNG
   RUNG wire#w1
      Contact( "FinalCutLub".COut.IsRunning )
      S_Coil( #MB2_Decoder.OpEnabled )
   END_RUNG
   RUNG wire#w1
      Contact( "FinalCutLub".COut.IsRunning )
      S_Coil( #MB2_Decoder.OpRunning )
   END_RUNG
   RUNG wire#w1
      Contact( "Sys".Bit0 )
      S_Coil( #MB2_Decoder.OpDone )
   END_RUNG
   // the same network as SCL:
   #_w1 := #MB2_Decoder.Code = #"2055_FINALCUT_LUBR";
   "A02_HMI".MB2.Button.FinalCut.Lubr.Stop := #_w1 AND #MB2_Decoder.OperationMinus;
   "A02_HMI".MB2.Button.FinalCut.Lubr.Start := #_w1 AND #MB2_Decoder.OperationPlus;
   IF #_w1 AND "FinalCutLub".COut.IsRunning THEN
       #MB2_Decoder.OpEnabled := TRUE;
       #MB2_Decoder.OpRunning := TRUE;
   END_IF;
   IF #_w1 AND "Sys".Bit0 THEN #MB2_Decoder.OpDone := TRUE; END_IF;
END_REGION

REGION Network 21: >
END_REGION

REGION Network 22: MB2 Code 2061 - AccDecConveyor ROLLS COMBO MOVE
   RUNG wire#powerrail
      { S7_Templates := "SrcType := Int" } EQ_Contact(in1 := #MB2_Decoder.Code, in2 := #"2061_ACCROLLCONVEYOR_COMBO_MOVE")
      wire#w1
      Contact( #MB2_Decoder.OperationMinus )
      Coil( "A02_HMI".MB2.Button.AccRollConveyor.MoveCombo.Bwd_Minus )
   END_RUNG
   RUNG wire#w1
      Contact( #MB2_Decoder.OperationPlus )
      Coil( "A02_HMI".MB2.Button.AccRollConveyor.MoveCombo.Fwd_Plus )
   END_RUNG
   RUNG wire#w1
      I_Contact( "AccRollConveyor".COut.Rolls.Fwd_CheckNext )
      I_Contact( "AccRollConveyor".COut.Rolls.Bwd_CheckNext )
      Not()
      S_Coil( #MB2_Decoder.OpEnabled )
   END_RUNG
   RUNG wire#w1
      I_Contact( "AccRollConveyor".COut.Rolls.Standstill )
      Contact( #MB2_Decoder.OpEnabled )
      S_Coil( #MB2_Decoder.OpRunning )
   END_RUNG
   RUNG wire#w1
      Contact( FALSE )
      S_Coil( #MB2_Decoder.OpDone )
   END_RUNG
   // the same network as SCL:
   #_w1 := #MB2_Decoder.Code = #"2061_ACCROLLCONVEYOR_COMBO_MOVE";
   "A02_HMI".MB2.Button.AccRollConveyor.MoveCombo.Bwd_Minus := #_w1 AND #MB2_Decoder.OperationMinus;
   "A02_HMI".MB2.Button.AccRollConveyor.MoveCombo.Fwd_Plus := #_w1 AND #MB2_Decoder.OperationPlus;
   IF NOT (#_w1 AND NOT "AccRollConveyor".COut.Rolls.Fwd_CheckNext AND NOT "AccRollConveyor".COut.Rolls.Bwd_CheckNext) THEN
       #MB2_Decoder.OpEnabled := TRUE;
   END_IF;
   IF #_w1 AND NOT "AccRollConveyor".COut.Rolls.Standstill AND #MB2_Decoder.OpEnabled THEN
       #MB2_Decoder.OpRunning := TRUE;
   END_IF;
   IF #_w1 AND FALSE THEN #MB2_Decoder.OpDone := TRUE; END_IF;
END_REGION

REGION Network 23: MB2 Code 2062 - AccDecConveyor PUSHER VERT COMBO
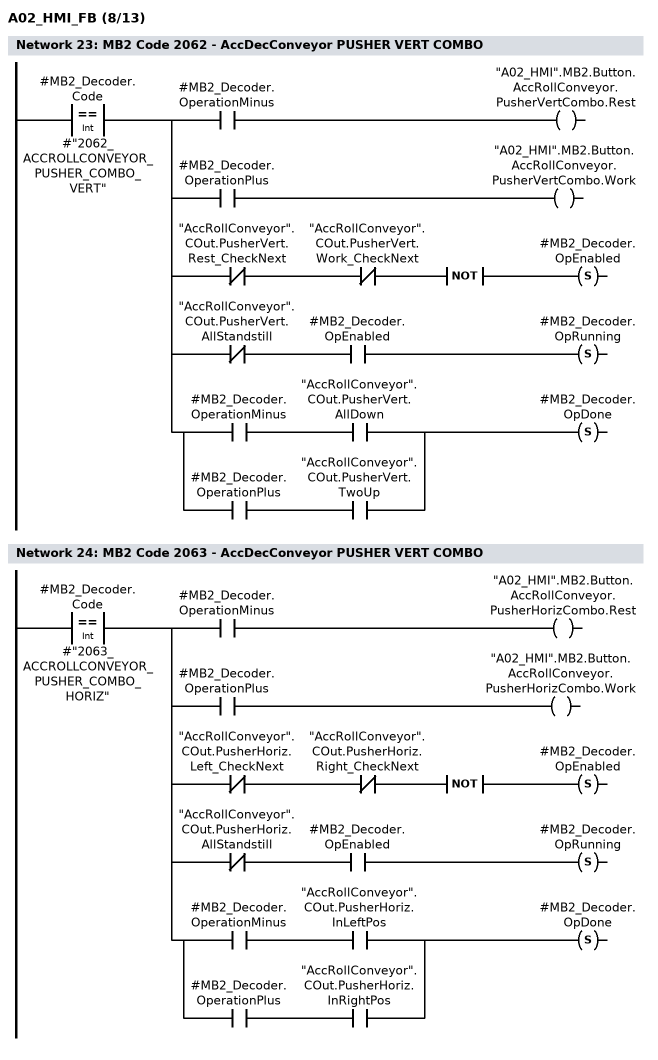
   RUNG wire#powerrail
      { S7_Templates := "SrcType := Int" } EQ_Contact(in1 := #MB2_Decoder.Code, in2 := #"2062_ACCROLLCONVEYOR_PUSHER_COMBO_VERT")
      wire#w1
      Contact( #MB2_Decoder.OperationMinus )
      Coil( "A02_HMI".MB2.Button.AccRollConveyor.PusherVertCombo.Rest )
   END_RUNG
   RUNG wire#w1
      Contact( #MB2_Decoder.OperationPlus )
      Coil( "A02_HMI".MB2.Button.AccRollConveyor.PusherVertCombo.Work )
   END_RUNG
   RUNG wire#w1
      I_Contact( "AccRollConveyor".COut.PusherVert.Rest_CheckNext )
      I_Contact( "AccRollConveyor".COut.PusherVert.Work_CheckNext )
      Not()
      S_Coil( #MB2_Decoder.OpEnabled )
   END_RUNG
   RUNG wire#w1
      I_Contact( "AccRollConveyor".COut.PusherVert.AllStandstill )
      Contact( #MB2_Decoder.OpEnabled )
      S_Coil( #MB2_Decoder.OpRunning )
   END_RUNG
   RUNG wire#w1
      Contact( #MB2_Decoder.OperationMinus )
      Contact( "AccRollConveyor".COut.PusherVert.AllDown )
      wire#w2
      S_Coil( #MB2_Decoder.OpDone )
   END_RUNG
   RUNG wire#w1
      Contact( #MB2_Decoder.OperationPlus )
      Contact( "AccRollConveyor".COut.PusherVert.TwoUp )
   END_RUNG wire#w2
   // the same network as SCL:
   #_w1 := #MB2_Decoder.Code = #"2062_ACCROLLCONVEYOR_PUSHER_COMBO_VERT";
   "A02_HMI".MB2.Button.AccRollConveyor.PusherVertCombo.Rest := #_w1 AND #MB2_Decoder.OperationMinus;
   "A02_HMI".MB2.Button.AccRollConveyor.PusherVertCombo.Work := #_w1 AND #MB2_Decoder.OperationPlus;
   IF NOT (#_w1 AND NOT "AccRollConveyor".COut.PusherVert.Rest_CheckNext AND NOT "AccRollConveyor".COut.PusherVert.Work_CheckNext) THEN
       #MB2_Decoder.OpEnabled := TRUE;
   END_IF;
   IF #_w1 AND NOT "AccRollConveyor".COut.PusherVert.AllStandstill AND #MB2_Decoder.OpEnabled THEN
       #MB2_Decoder.OpRunning := TRUE;
   END_IF;
   IF #_w1 AND ((#MB2_Decoder.OperationMinus AND "AccRollConveyor".COut.PusherVert.AllDown) OR (#MB2_Decoder.OperationPlus AND "AccRollConveyor".COut.PusherVert.TwoUp)) THEN
       #MB2_Decoder.OpDone := TRUE;
   END_IF;
END_REGION

REGION Network 24: MB2 Code 2063 - AccDecConveyor PUSHER VERT COMBO
   RUNG wire#powerrail
      { S7_Templates := "SrcType := Int" } EQ_Contact(in1 := #MB2_Decoder.Code, in2 := #"2063_ACCROLLCONVEYOR_PUSHER_COMBO_HORIZ")
      wire#w1
      Contact( #MB2_Decoder.OperationMinus )
      Coil( "A02_HMI".MB2.Button.AccRollConveyor.PusherHorizCombo.Rest )
   END_RUNG
   RUNG wire#w1
      Contact( #MB2_Decoder.OperationPlus )
      Coil( "A02_HMI".MB2.Button.AccRollConveyor.PusherHorizCombo.Work )
   END_RUNG
   RUNG wire#w1
      I_Contact( "AccRollConveyor".COut.PusherHoriz.Left_CheckNext )
      I_Contact( "AccRollConveyor".COut.PusherHoriz.Right_CheckNext )
      Not()
      S_Coil( #MB2_Decoder.OpEnabled )
   END_RUNG
   RUNG wire#w1
      I_Contact( "AccRollConveyor".COut.PusherHoriz.AllStandstill )
      Contact( #MB2_Decoder.OpEnabled )
      S_Coil( #MB2_Decoder.OpRunning )
   END_RUNG
   RUNG wire#w1
      Contact( #MB2_Decoder.OperationMinus )
      Contact( "AccRollConveyor".COut.PusherHoriz.InLeftPos )
      wire#w2
      S_Coil( #MB2_Decoder.OpDone )
   END_RUNG
   RUNG wire#w1
      Contact( #MB2_Decoder.OperationPlus )
      Contact( "AccRollConveyor".COut.PusherHoriz.InRightPos )
   END_RUNG wire#w2
   // the same network as SCL:
   #_w1 := #MB2_Decoder.Code = #"2063_ACCROLLCONVEYOR_PUSHER_COMBO_HORIZ";
   "A02_HMI".MB2.Button.AccRollConveyor.PusherHorizCombo.Rest := #_w1 AND #MB2_Decoder.OperationMinus;
   "A02_HMI".MB2.Button.AccRollConveyor.PusherHorizCombo.Work := #_w1 AND #MB2_Decoder.OperationPlus;
   IF NOT (#_w1 AND NOT "AccRollConveyor".COut.PusherHoriz.Left_CheckNext AND NOT "AccRollConveyor".COut.PusherHoriz.Right_CheckNext) THEN
       #MB2_Decoder.OpEnabled := TRUE;
   END_IF;
   IF #_w1 AND NOT "AccRollConveyor".COut.PusherHoriz.AllStandstill AND #MB2_Decoder.OpEnabled THEN
       #MB2_Decoder.OpRunning := TRUE;
   END_IF;
   IF #_w1 AND ((#MB2_Decoder.OperationMinus AND "AccRollConveyor".COut.PusherHoriz.InLeftPos) OR (#MB2_Decoder.OperationPlus AND "AccRollConveyor".COut.PusherHoriz.InRightPos)) THEN
       #MB2_Decoder.OpDone := TRUE;
   END_IF;
END_REGION

REGION Network 25: MB2 Code 2071 - AccDecConveyor ROLLS 1
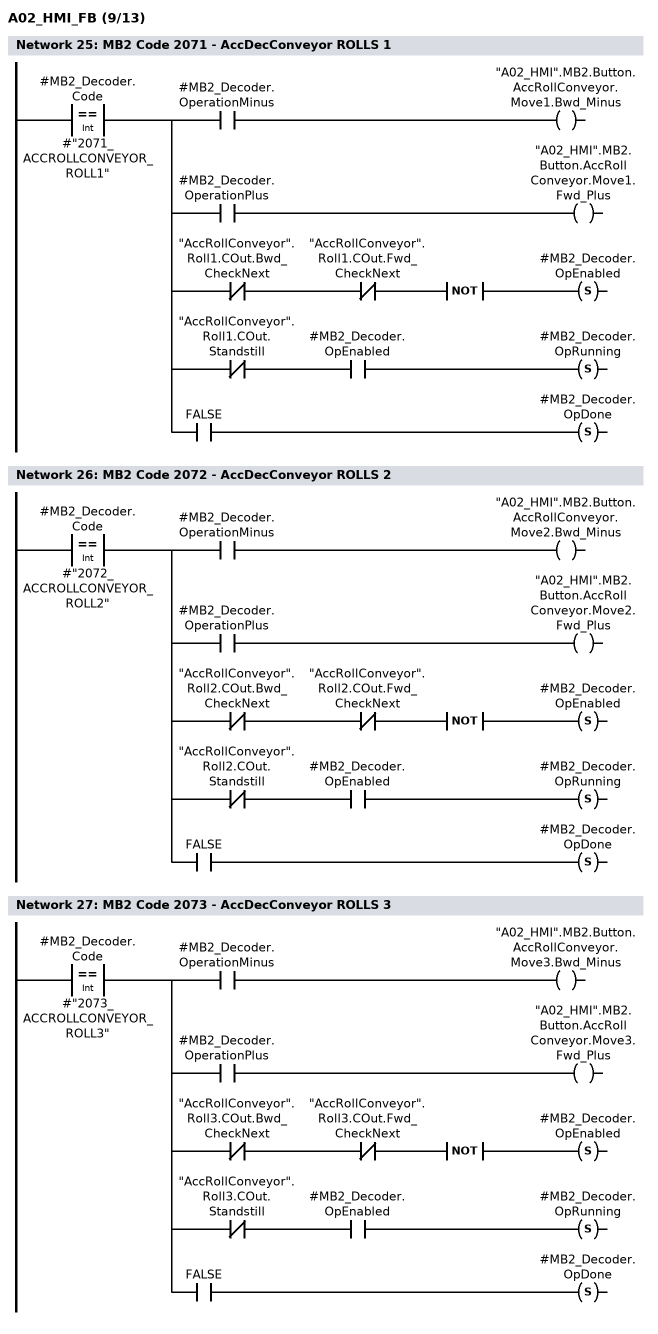
   RUNG wire#powerrail
      { S7_Templates := "SrcType := Int" } EQ_Contact(in1 := #MB2_Decoder.Code, in2 := #"2071_ACCROLLCONVEYOR_ROLL1")
      wire#w1
      Contact( #MB2_Decoder.OperationMinus )
      Coil( "A02_HMI".MB2.Button.AccRollConveyor.Move1.Bwd_Minus )
   END_RUNG
   RUNG wire#w1
      Contact( #MB2_Decoder.OperationPlus )
      Coil( "A02_HMI".MB2.Button.AccRollConveyor.Move1.Fwd_Plus )
   END_RUNG
   RUNG wire#w1
      I_Contact( "AccRollConveyor".Roll1.COut.Bwd_CheckNext )
      I_Contact( "AccRollConveyor".Roll1.COut.Fwd_CheckNext )
      Not()
      S_Coil( #MB2_Decoder.OpEnabled )
   END_RUNG
   RUNG wire#w1
      I_Contact( "AccRollConveyor".Roll1.COut.Standstill )
      Contact( #MB2_Decoder.OpEnabled )
      S_Coil( #MB2_Decoder.OpRunning )
   END_RUNG
   RUNG wire#w1
      Contact( FALSE )
      S_Coil( #MB2_Decoder.OpDone )
   END_RUNG
   // the same network as SCL:
   #_w1 := #MB2_Decoder.Code = #"2071_ACCROLLCONVEYOR_ROLL1";
   "A02_HMI".MB2.Button.AccRollConveyor.Move1.Bwd_Minus := #_w1 AND #MB2_Decoder.OperationMinus;
   "A02_HMI".MB2.Button.AccRollConveyor.Move1.Fwd_Plus := #_w1 AND #MB2_Decoder.OperationPlus;
   IF NOT (#_w1 AND NOT "AccRollConveyor".Roll1.COut.Bwd_CheckNext AND NOT "AccRollConveyor".Roll1.COut.Fwd_CheckNext) THEN
       #MB2_Decoder.OpEnabled := TRUE;
   END_IF;
   IF #_w1 AND NOT "AccRollConveyor".Roll1.COut.Standstill AND #MB2_Decoder.OpEnabled THEN
       #MB2_Decoder.OpRunning := TRUE;
   END_IF;
   IF #_w1 AND FALSE THEN #MB2_Decoder.OpDone := TRUE; END_IF;
END_REGION

REGION Network 26: MB2 Code 2072 - AccDecConveyor ROLLS 2
   RUNG wire#powerrail
      { S7_Templates := "SrcType := Int" } EQ_Contact(in1 := #MB2_Decoder.Code, in2 := #"2072_ACCROLLCONVEYOR_ROLL2")
      wire#w1
      Contact( #MB2_Decoder.OperationMinus )
      Coil( "A02_HMI".MB2.Button.AccRollConveyor.Move2.Bwd_Minus )
   END_RUNG
   RUNG wire#w1
      Contact( #MB2_Decoder.OperationPlus )
      Coil( "A02_HMI".MB2.Button.AccRollConveyor.Move2.Fwd_Plus )
   END_RUNG
   RUNG wire#w1
      I_Contact( "AccRollConveyor".Roll2.COut.Bwd_CheckNext )
      I_Contact( "AccRollConveyor".Roll2.COut.Fwd_CheckNext )
      Not()
      S_Coil( #MB2_Decoder.OpEnabled )
   END_RUNG
   RUNG wire#w1
      I_Contact( "AccRollConveyor".Roll2.COut.Standstill )
      Contact( #MB2_Decoder.OpEnabled )
      S_Coil( #MB2_Decoder.OpRunning )
   END_RUNG
   RUNG wire#w1
      Contact( FALSE )
      S_Coil( #MB2_Decoder.OpDone )
   END_RUNG
   // the same network as SCL:
   #_w1 := #MB2_Decoder.Code = #"2072_ACCROLLCONVEYOR_ROLL2";
   "A02_HMI".MB2.Button.AccRollConveyor.Move2.Bwd_Minus := #_w1 AND #MB2_Decoder.OperationMinus;
   "A02_HMI".MB2.Button.AccRollConveyor.Move2.Fwd_Plus := #_w1 AND #MB2_Decoder.OperationPlus;
   IF NOT (#_w1 AND NOT "AccRollConveyor".Roll2.COut.Bwd_CheckNext AND NOT "AccRollConveyor".Roll2.COut.Fwd_CheckNext) THEN
       #MB2_Decoder.OpEnabled := TRUE;
   END_IF;
   IF #_w1 AND NOT "AccRollConveyor".Roll2.COut.Standstill AND #MB2_Decoder.OpEnabled THEN
       #MB2_Decoder.OpRunning := TRUE;
   END_IF;
   IF #_w1 AND FALSE THEN #MB2_Decoder.OpDone := TRUE; END_IF;
END_REGION

REGION Network 27: MB2 Code 2073 - AccDecConveyor ROLLS 3
   RUNG wire#powerrail
      { S7_Templates := "SrcType := Int" } EQ_Contact(in1 := #MB2_Decoder.Code, in2 := #"2073_ACCROLLCONVEYOR_ROLL3")
      wire#w1
      Contact( #MB2_Decoder.OperationMinus )
      Coil( "A02_HMI".MB2.Button.AccRollConveyor.Move3.Bwd_Minus )
   END_RUNG
   RUNG wire#w1
      Contact( #MB2_Decoder.OperationPlus )
      Coil( "A02_HMI".MB2.Button.AccRollConveyor.Move3.Fwd_Plus )
   END_RUNG
   RUNG wire#w1
      I_Contact( "AccRollConveyor".Roll3.COut.Bwd_CheckNext )
      I_Contact( "AccRollConveyor".Roll3.COut.Fwd_CheckNext )
      Not()
      S_Coil( #MB2_Decoder.OpEnabled )
   END_RUNG
   RUNG wire#w1
      I_Contact( "AccRollConveyor".Roll3.COut.Standstill )
      Contact( #MB2_Decoder.OpEnabled )
      S_Coil( #MB2_Decoder.OpRunning )
   END_RUNG
   RUNG wire#w1
      Contact( FALSE )
      S_Coil( #MB2_Decoder.OpDone )
   END_RUNG
   // the same network as SCL:
   #_w1 := #MB2_Decoder.Code = #"2073_ACCROLLCONVEYOR_ROLL3";
   "A02_HMI".MB2.Button.AccRollConveyor.Move3.Bwd_Minus := #_w1 AND #MB2_Decoder.OperationMinus;
   "A02_HMI".MB2.Button.AccRollConveyor.Move3.Fwd_Plus := #_w1 AND #MB2_Decoder.OperationPlus;
   IF NOT (#_w1 AND NOT "AccRollConveyor".Roll3.COut.Bwd_CheckNext AND NOT "AccRollConveyor".Roll3.COut.Fwd_CheckNext) THEN
       #MB2_Decoder.OpEnabled := TRUE;
   END_IF;
   IF #_w1 AND NOT "AccRollConveyor".Roll3.COut.Standstill AND #MB2_Decoder.OpEnabled THEN
       #MB2_Decoder.OpRunning := TRUE;
   END_IF;
   IF #_w1 AND FALSE THEN #MB2_Decoder.OpDone := TRUE; END_IF;
END_REGION

REGION Network 29 (SCL): MB2 Code 2081 ... PUSHER SINGLE


   FOR #i := 1 TO "MAX_PUSHER" DO

       "A02_HMI".MB2.Button.AccRollConveyor.PusherVert_Single[#i].Rest := FALSE;
       "A02_HMI".MB2.Button.AccRollConveyor.PusherVert_Single[#i].Work := FALSE;
       "A02_HMI".MB2.Button.AccRollConveyor.PusherVert_Single[#i].Work := FALSE;

       "A02_HMI".MB2.Button.AccRollConveyor.PusherHoriz_Single[#i].Rest := FALSE;
       "A02_HMI".MB2.Button.AccRollConveyor.PusherHoriz_Single[#i].Work := FALSE;
       "A02_HMI".MB2.Button.AccRollConveyor.PusherHoriz_Single[#i].Work := FALSE;

       #tempIdxVert := #"2081_ACCROLLCONVEYOR_PUSHER_VERT_1" + (#i - 1);
       #tempIdxHoriz := #"2091_ACCROLLCONVEYOR_PUSHER_HORIZ_1" + (#i - 1);

       IF #MB2_Decoder.Code = #tempIdxVert THEN

           "A02_HMI".MB2.Button.AccRollConveyor.PusherVert_Single[#i].Rest := #MB2_Decoder.OperationMinus;
           "A02_HMI".MB2.Button.AccRollConveyor.PusherVert_Single[#i].Work := #MB2_Decoder.OperationPlus;

           #MB2_Decoder.OpEnabled := "AccRollConveyor".PusherVert[#i].COut.Rest_CheckNext OR "AccRollConveyor".PusherVert[#i].COut.Work_CheckNext;
           #MB2_Decoder.OpRunning := "AccRollConveyor".PusherVert[#i].COut.Standstill AND #MB2_Decoder.OpEnabled;
           #MB2_Decoder.OpDone := (#MB2_Decoder.OperationMinus AND "AccRollConveyor".PusherVert[#i].COut.Rest) OR (#MB2_Decoder.OperationPlus AND "AccRollConveyor".PusherVert[#i].COut.Work);

       END_IF;

       IF #MB2_Decoder.Code = #tempIdxHoriz THEN

           "A02_HMI".MB2.Button.AccRollConveyor.PusherHoriz_Single[#i].Rest := #MB2_Decoder.OperationMinus;
           "A02_HMI".MB2.Button.AccRollConveyor.PusherHoriz_Single[#i].Work := #MB2_Decoder.OperationPlus;

           #MB2_Decoder.OpEnabled := "AccRollConveyor".PusherHoriz[#i].COut.Rest_CheckNext OR "AccRollConveyor".PusherHoriz[#i].COut.Work_CheckNext;
           #MB2_Decoder.OpRunning := "AccRollConveyor".PusherHoriz[#i].COut.Standstill AND #MB2_Decoder.OpEnabled;
           #MB2_Decoder.OpDone := (#MB2_Decoder.OperationMinus AND "AccRollConveyor".PusherHoriz[#i].COut.Rest) OR (#MB2_Decoder.OperationPlus AND "AccRollConveyor".PusherHoriz[#i].COut.Work);

       END_IF;


   END_FOR;
END_REGION

REGION Network 30: >
END_REGION

REGION Network 31 (SCL): MB2 Code REGOLAZIONE FORMATO

   FOR #i := 1 TO 14 DO

       "A02_HMI".MB2.Button.Profilatrice_RegolazioneFormato.Single_PB[#i].Bwd_Minus := FALSE;
       "A02_HMI".MB2.Button.Profilatrice_RegolazioneFormato.Single_PB[#i].Fwd_Plus := FALSE;
       "A02_HMI".MB2.Button.Profilatrice_RegolazioneFormato.Single_PB[#i].MoveToPos := FALSE;

       #tempIdxMove := #"2100_MODULO1_OP_MOVE" + ((#i - 1) * 2);
       #tempIdxPos := #"2101_MODULO1_OP_POS" + ((#i - 1) * 2);

       IF #MB2_Decoder.Code = #tempIdxMove THEN

           "A02_HMI".MB2.Button.Profilatrice_RegolazioneFormato.Single_PB[#i].Bwd_Minus := #MB2_Decoder.OperationMinus;
           "A02_HMI".MB2.Button.Profilatrice_RegolazioneFormato.Single_PB[#i].Fwd_Plus := #MB2_Decoder.OperationPlus;

           IF #i <= 6 THEN
               #MB2_Decoder.OpEnabled := "A0201_Profilatrice_RegolazioneFormato".AX_D[#i].COut.MinusCheckNext OR "A0201_Profilatrice_RegolazioneFormato".AX_D[#i].COut.PlusCheckNext;
               #MB2_Decoder.OpRunning := NOT "A0201_Profilatrice_RegolazioneFormato".AX_D[#i].COut.Standstill AND #MB2_Decoder.OpEnabled;
               #MB2_Decoder.OpDone := "A0201_Profilatrice_RegolazioneFormato".AX_D[#i].COut.PlusLimitReached OR "A0201_Profilatrice_RegolazioneFormato".AX_D[#i].COut.MinusLimitReached OR "A0201_Profilatrice_RegolazioneFormato".AX_D[#i].COut.InPosition;
           ELSE
               #MB2_Decoder.OpEnabled := "A0201_Profilatrice_RegolazioneFormato".AX_M[#i].COut.MinusCheckNext OR "A0201_Profilatrice_RegolazioneFormato".AX_M[#i].COut.PlusCheckNext;
               #MB2_Decoder.OpRunning := NOT "A0201_Profilatrice_RegolazioneFormato".AX_M[#i].COut.Standstill AND #MB2_Decoder.OpEnabled;
               #MB2_Decoder.OpDone := "A0201_Profilatrice_RegolazioneFormato".AX_M[#i].COut.PlusLimitReached OR "A0201_Profilatrice_RegolazioneFormato".AX_M[#i].COut.MinusLimitReached OR "A0201_Profilatrice_RegolazioneFormato".AX_M[#i].COut.InPosition;
           END_IF;

       ELSIF #MB2_Decoder.Code = #tempIdxPos THEN
           "A02_HMI".MB2.Button.Profilatrice_RegolazioneFormato.Single_PB[#i].MoveToPos := #MB2_Decoder.OperationPlus;

           IF #i <= 6 THEN
               #MB2_Decoder.OpEnabled := "A0201_Profilatrice_RegolazioneFormato".AX_D[#i].COut.MinusCheckNext OR "A0201_Profilatrice_RegolazioneFormato".AX_D[#i].COut.PlusCheckNext;
               #MB2_Decoder.OpRunning := NOT "A0201_Profilatrice_RegolazioneFormato".AX_D[#i].COut.Standstill AND #MB2_Decoder.OpEnabled;
               #MB2_Decoder.OpDone :=  "A0201_Profilatrice_RegolazioneFormato".AX_D[#i].COut.InPosition;
           ELSE
               #MB2_Decoder.OpEnabled := "A0201_Profilatrice_RegolazioneFormato".AX_M[#i].COut.MinusCheckNext OR "A0201_Profilatrice_RegolazioneFormato".AX_M[#i].COut.PlusCheckNext;
               #MB2_Decoder.OpRunning := NOT "A0201_Profilatrice_RegolazioneFormato".AX_M[#i].COut.Standstill AND #MB2_Decoder.OpEnabled;
               #MB2_Decoder.OpDone := "A0201_Profilatrice_RegolazioneFormato".AX_M[#i].COut.InPosition;
           END_IF;


       END_IF;


   END_FOR;
END_REGION

REGION Network 32: MB2 Code 2280_PASSAGGIO2_COMBO_MOVE
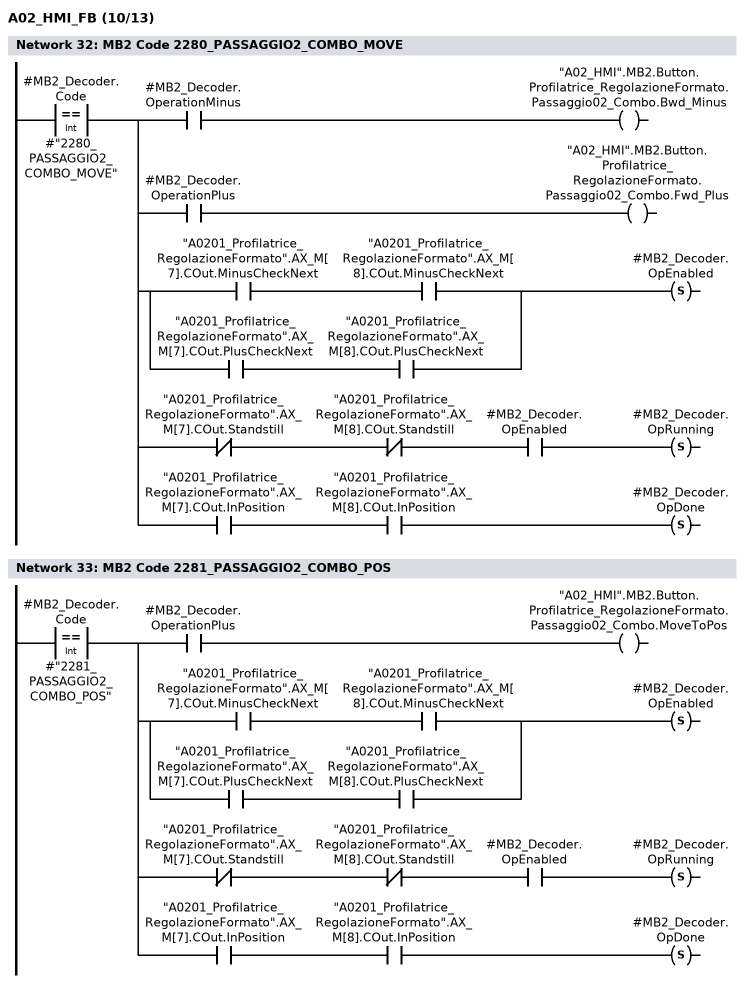
   RUNG wire#powerrail
      { S7_Templates := "SrcType := Int" } EQ_Contact(in1 := #MB2_Decoder.Code, in2 := #"2280_PASSAGGIO2_COMBO_MOVE")
      wire#w1
      Contact( #MB2_Decoder.OperationMinus )
      Coil( "A02_HMI".MB2.Button.Profilatrice_RegolazioneFormato.Passaggio02_Combo.Bwd_Minus )
   END_RUNG
   RUNG wire#w1
      Contact( #MB2_Decoder.OperationPlus )
      Coil( "A02_HMI".MB2.Button.Profilatrice_RegolazioneFormato.Passaggio02_Combo.Fwd_Plus )
   END_RUNG
   RUNG wire#w1
      Contact( "A0201_Profilatrice_RegolazioneFormato".AX_M[7].COut.MinusCheckNext )
      Contact( "A0201_Profilatrice_RegolazioneFormato".AX_M[8].COut.MinusCheckNext )
      wire#w2
      S_Coil( #MB2_Decoder.OpEnabled )
   END_RUNG
   RUNG wire#w1
      Contact( "A0201_Profilatrice_RegolazioneFormato".AX_M[7].COut.PlusCheckNext )
      Contact( "A0201_Profilatrice_RegolazioneFormato".AX_M[8].COut.PlusCheckNext )
   END_RUNG wire#w2
   RUNG wire#w1
      I_Contact( "A0201_Profilatrice_RegolazioneFormato".AX_M[7].COut.Standstill )
      I_Contact( "A0201_Profilatrice_RegolazioneFormato".AX_M[8].COut.Standstill )
      Contact( #MB2_Decoder.OpEnabled )
      S_Coil( #MB2_Decoder.OpRunning )
   END_RUNG
   RUNG wire#w1
      Contact( "A0201_Profilatrice_RegolazioneFormato".AX_M[7].COut.InPosition )
      Contact( "A0201_Profilatrice_RegolazioneFormato".AX_M[8].COut.InPosition )
      S_Coil( #MB2_Decoder.OpDone )
   END_RUNG
   // the same network as SCL:
   #_w1 := #MB2_Decoder.Code = #"2280_PASSAGGIO2_COMBO_MOVE";
   "A02_HMI".MB2.Button.Profilatrice_RegolazioneFormato.Passaggio02_Combo.Bwd_Minus := #_w1 AND #MB2_Decoder.OperationMinus;
   "A02_HMI".MB2.Button.Profilatrice_RegolazioneFormato.Passaggio02_Combo.Fwd_Plus := #_w1 AND #MB2_Decoder.OperationPlus;
   IF #_w1 AND (("A0201_Profilatrice_RegolazioneFormato".AX_M[7].COut.MinusCheckNext AND "A0201_Profilatrice_RegolazioneFormato".AX_M[8].COut.MinusCheckNext) OR ("A0201_Profilatrice_RegolazioneFormato".AX_M[7].COut.PlusCheckNext AND "A0201_Profilatrice_RegolazioneFormato".AX_M[8].COut.PlusCheckNext)) THEN
       #MB2_Decoder.OpEnabled := TRUE;
   END_IF;
   IF #_w1 AND NOT "A0201_Profilatrice_RegolazioneFormato".AX_M[7].COut.Standstill AND NOT "A0201_Profilatrice_RegolazioneFormato".AX_M[8].COut.Standstill AND #MB2_Decoder.OpEnabled THEN
       #MB2_Decoder.OpRunning := TRUE;
   END_IF;
   IF #_w1 AND "A0201_Profilatrice_RegolazioneFormato".AX_M[7].COut.InPosition AND "A0201_Profilatrice_RegolazioneFormato".AX_M[8].COut.InPosition THEN
       #MB2_Decoder.OpDone := TRUE;
   END_IF;
END_REGION

REGION Network 33: MB2 Code 2281_PASSAGGIO2_COMBO_POS
   RUNG wire#powerrail
      { S7_Templates := "SrcType := Int" } EQ_Contact(in1 := #MB2_Decoder.Code, in2 := #"2281_PASSAGGIO2_COMBO_POS")
      wire#w1
      Contact( #MB2_Decoder.OperationPlus )
      Coil( "A02_HMI".MB2.Button.Profilatrice_RegolazioneFormato.Passaggio02_Combo.MoveToPos )
   END_RUNG
   RUNG wire#w1
      Contact( "A0201_Profilatrice_RegolazioneFormato".AX_M[7].COut.MinusCheckNext )
      Contact( "A0201_Profilatrice_RegolazioneFormato".AX_M[8].COut.MinusCheckNext )
      wire#w2
      S_Coil( #MB2_Decoder.OpEnabled )
   END_RUNG
   RUNG wire#w1
      Contact( "A0201_Profilatrice_RegolazioneFormato".AX_M[7].COut.PlusCheckNext )
      Contact( "A0201_Profilatrice_RegolazioneFormato".AX_M[8].COut.PlusCheckNext )
   END_RUNG wire#w2
   RUNG wire#w1
      I_Contact( "A0201_Profilatrice_RegolazioneFormato".AX_M[7].COut.Standstill )
      I_Contact( "A0201_Profilatrice_RegolazioneFormato".AX_M[8].COut.Standstill )
      Contact( #MB2_Decoder.OpEnabled )
      S_Coil( #MB2_Decoder.OpRunning )
   END_RUNG
   RUNG wire#w1
      Contact( "A0201_Profilatrice_RegolazioneFormato".AX_M[7].COut.InPosition )
      Contact( "A0201_Profilatrice_RegolazioneFormato".AX_M[8].COut.InPosition )
      S_Coil( #MB2_Decoder.OpDone )
   END_RUNG
   // the same network as SCL:
   #_w1 := #MB2_Decoder.Code = #"2281_PASSAGGIO2_COMBO_POS";
   "A02_HMI".MB2.Button.Profilatrice_RegolazioneFormato.Passaggio02_Combo.MoveToPos := #_w1 AND #MB2_Decoder.OperationPlus;
   IF #_w1 AND (("A0201_Profilatrice_RegolazioneFormato".AX_M[7].COut.MinusCheckNext AND "A0201_Profilatrice_RegolazioneFormato".AX_M[8].COut.MinusCheckNext) OR ("A0201_Profilatrice_RegolazioneFormato".AX_M[7].COut.PlusCheckNext AND "A0201_Profilatrice_RegolazioneFormato".AX_M[8].COut.PlusCheckNext)) THEN
       #MB2_Decoder.OpEnabled := TRUE;
   END_IF;
   IF #_w1 AND NOT "A0201_Profilatrice_RegolazioneFormato".AX_M[7].COut.Standstill AND NOT "A0201_Profilatrice_RegolazioneFormato".AX_M[8].COut.Standstill AND #MB2_Decoder.OpEnabled THEN
       #MB2_Decoder.OpRunning := TRUE;
   END_IF;
   IF #_w1 AND "A0201_Profilatrice_RegolazioneFormato".AX_M[7].COut.InPosition AND "A0201_Profilatrice_RegolazioneFormato".AX_M[8].COut.InPosition THEN
       #MB2_Decoder.OpDone := TRUE;
   END_IF;
END_REGION

REGION Network 34: MB2 Code 2282_PASSAGGIO14_COMBO_MOVE
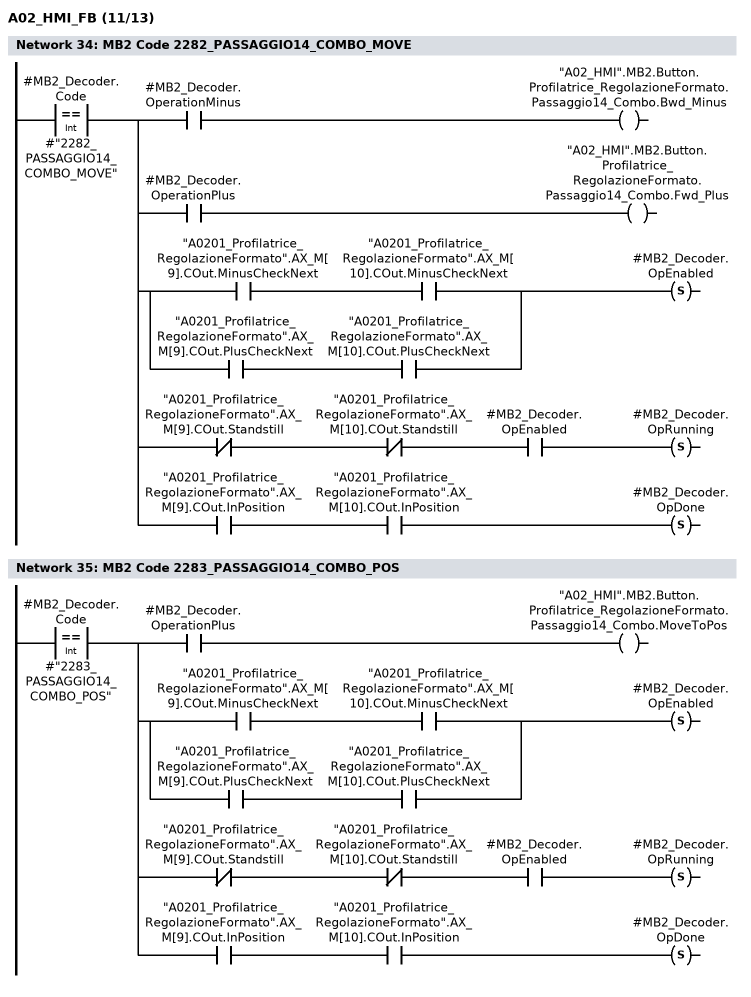
   RUNG wire#powerrail
      { S7_Templates := "SrcType := Int" } EQ_Contact(in1 := #MB2_Decoder.Code, in2 := #"2282_PASSAGGIO14_COMBO_MOVE")
      wire#w1
      Contact( #MB2_Decoder.OperationMinus )
      Coil( "A02_HMI".MB2.Button.Profilatrice_RegolazioneFormato.Passaggio14_Combo.Bwd_Minus )
   END_RUNG
   RUNG wire#w1
      Contact( #MB2_Decoder.OperationPlus )
      Coil( "A02_HMI".MB2.Button.Profilatrice_RegolazioneFormato.Passaggio14_Combo.Fwd_Plus )
   END_RUNG
   RUNG wire#w1
      Contact( "A0201_Profilatrice_RegolazioneFormato".AX_M[9].COut.MinusCheckNext )
      Contact( "A0201_Profilatrice_RegolazioneFormato".AX_M[10].COut.MinusCheckNext )
      wire#w2
      S_Coil( #MB2_Decoder.OpEnabled )
   END_RUNG
   RUNG wire#w1
      Contact( "A0201_Profilatrice_RegolazioneFormato".AX_M[9].COut.PlusCheckNext )
      Contact( "A0201_Profilatrice_RegolazioneFormato".AX_M[10].COut.PlusCheckNext )
   END_RUNG wire#w2
   RUNG wire#w1
      I_Contact( "A0201_Profilatrice_RegolazioneFormato".AX_M[9].COut.Standstill )
      I_Contact( "A0201_Profilatrice_RegolazioneFormato".AX_M[10].COut.Standstill )
      Contact( #MB2_Decoder.OpEnabled )
      S_Coil( #MB2_Decoder.OpRunning )
   END_RUNG
   RUNG wire#w1
      Contact( "A0201_Profilatrice_RegolazioneFormato".AX_M[9].COut.InPosition )
      Contact( "A0201_Profilatrice_RegolazioneFormato".AX_M[10].COut.InPosition )
      S_Coil( #MB2_Decoder.OpDone )
   END_RUNG
   // the same network as SCL:
   #_w1 := #MB2_Decoder.Code = #"2282_PASSAGGIO14_COMBO_MOVE";
   "A02_HMI".MB2.Button.Profilatrice_RegolazioneFormato.Passaggio14_Combo.Bwd_Minus := #_w1 AND #MB2_Decoder.OperationMinus;
   "A02_HMI".MB2.Button.Profilatrice_RegolazioneFormato.Passaggio14_Combo.Fwd_Plus := #_w1 AND #MB2_Decoder.OperationPlus;
   IF #_w1 AND (("A0201_Profilatrice_RegolazioneFormato".AX_M[9].COut.MinusCheckNext AND "A0201_Profilatrice_RegolazioneFormato".AX_M[10].COut.MinusCheckNext) OR ("A0201_Profilatrice_RegolazioneFormato".AX_M[9].COut.PlusCheckNext AND "A0201_Profilatrice_RegolazioneFormato".AX_M[10].COut.PlusCheckNext)) THEN
       #MB2_Decoder.OpEnabled := TRUE;
   END_IF;
   IF #_w1 AND NOT "A0201_Profilatrice_RegolazioneFormato".AX_M[9].COut.Standstill AND NOT "A0201_Profilatrice_RegolazioneFormato".AX_M[10].COut.Standstill AND #MB2_Decoder.OpEnabled THEN
       #MB2_Decoder.OpRunning := TRUE;
   END_IF;
   IF #_w1 AND "A0201_Profilatrice_RegolazioneFormato".AX_M[9].COut.InPosition AND "A0201_Profilatrice_RegolazioneFormato".AX_M[10].COut.InPosition THEN
       #MB2_Decoder.OpDone := TRUE;
   END_IF;
END_REGION

REGION Network 35: MB2 Code 2283_PASSAGGIO14_COMBO_POS
   RUNG wire#powerrail
      { S7_Templates := "SrcType := Int" } EQ_Contact(in1 := #MB2_Decoder.Code, in2 := #"2283_PASSAGGIO14_COMBO_POS")
      wire#w1
      Contact( #MB2_Decoder.OperationPlus )
      Coil( "A02_HMI".MB2.Button.Profilatrice_RegolazioneFormato.Passaggio14_Combo.MoveToPos )
   END_RUNG
   RUNG wire#w1
      Contact( "A0201_Profilatrice_RegolazioneFormato".AX_M[9].COut.MinusCheckNext )
      Contact( "A0201_Profilatrice_RegolazioneFormato".AX_M[10].COut.MinusCheckNext )
      wire#w2
      S_Coil( #MB2_Decoder.OpEnabled )
   END_RUNG
   RUNG wire#w1
      Contact( "A0201_Profilatrice_RegolazioneFormato".AX_M[9].COut.PlusCheckNext )
      Contact( "A0201_Profilatrice_RegolazioneFormato".AX_M[10].COut.PlusCheckNext )
   END_RUNG wire#w2
   RUNG wire#w1
      I_Contact( "A0201_Profilatrice_RegolazioneFormato".AX_M[9].COut.Standstill )
      I_Contact( "A0201_Profilatrice_RegolazioneFormato".AX_M[10].COut.Standstill )
      Contact( #MB2_Decoder.OpEnabled )
      S_Coil( #MB2_Decoder.OpRunning )
   END_RUNG
   RUNG wire#w1
      Contact( "A0201_Profilatrice_RegolazioneFormato".AX_M[9].COut.InPosition )
      Contact( "A0201_Profilatrice_RegolazioneFormato".AX_M[10].COut.InPosition )
      S_Coil( #MB2_Decoder.OpDone )
   END_RUNG
   // the same network as SCL:
   #_w1 := #MB2_Decoder.Code = #"2283_PASSAGGIO14_COMBO_POS";
   "A02_HMI".MB2.Button.Profilatrice_RegolazioneFormato.Passaggio14_Combo.MoveToPos := #_w1 AND #MB2_Decoder.OperationPlus;
   IF #_w1 AND (("A0201_Profilatrice_RegolazioneFormato".AX_M[9].COut.MinusCheckNext AND "A0201_Profilatrice_RegolazioneFormato".AX_M[10].COut.MinusCheckNext) OR ("A0201_Profilatrice_RegolazioneFormato".AX_M[9].COut.PlusCheckNext AND "A0201_Profilatrice_RegolazioneFormato".AX_M[10].COut.PlusCheckNext)) THEN
       #MB2_Decoder.OpEnabled := TRUE;
   END_IF;
   IF #_w1 AND NOT "A0201_Profilatrice_RegolazioneFormato".AX_M[9].COut.Standstill AND NOT "A0201_Profilatrice_RegolazioneFormato".AX_M[10].COut.Standstill AND #MB2_Decoder.OpEnabled THEN
       #MB2_Decoder.OpRunning := TRUE;
   END_IF;
   IF #_w1 AND "A0201_Profilatrice_RegolazioneFormato".AX_M[9].COut.InPosition AND "A0201_Profilatrice_RegolazioneFormato".AX_M[10].COut.InPosition THEN
       #MB2_Decoder.OpDone := TRUE;
   END_IF;
END_REGION

REGION Network 36: MB2 Code 2284_PASSAGGIO17_COMBO_MOVE
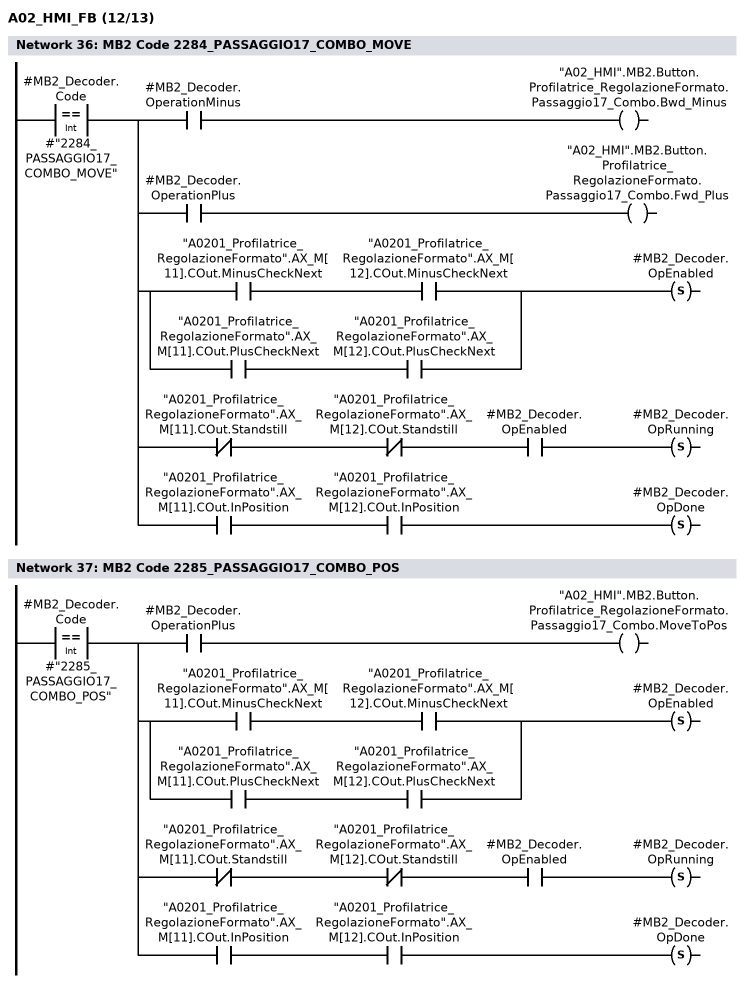
   RUNG wire#powerrail
      { S7_Templates := "SrcType := Int" } EQ_Contact(in1 := #MB2_Decoder.Code, in2 := #"2284_PASSAGGIO17_COMBO_MOVE")
      wire#w1
      Contact( #MB2_Decoder.OperationMinus )
      Coil( "A02_HMI".MB2.Button.Profilatrice_RegolazioneFormato.Passaggio17_Combo.Bwd_Minus )
   END_RUNG
   RUNG wire#w1
      Contact( #MB2_Decoder.OperationPlus )
      Coil( "A02_HMI".MB2.Button.Profilatrice_RegolazioneFormato.Passaggio17_Combo.Fwd_Plus )
   END_RUNG
   RUNG wire#w1
      Contact( "A0201_Profilatrice_RegolazioneFormato".AX_M[11].COut.MinusCheckNext )
      Contact( "A0201_Profilatrice_RegolazioneFormato".AX_M[12].COut.MinusCheckNext )
      wire#w2
      S_Coil( #MB2_Decoder.OpEnabled )
   END_RUNG
   RUNG wire#w1
      Contact( "A0201_Profilatrice_RegolazioneFormato".AX_M[11].COut.PlusCheckNext )
      Contact( "A0201_Profilatrice_RegolazioneFormato".AX_M[12].COut.PlusCheckNext )
   END_RUNG wire#w2
   RUNG wire#w1
      I_Contact( "A0201_Profilatrice_RegolazioneFormato".AX_M[11].COut.Standstill )
      I_Contact( "A0201_Profilatrice_RegolazioneFormato".AX_M[12].COut.Standstill )
      Contact( #MB2_Decoder.OpEnabled )
      S_Coil( #MB2_Decoder.OpRunning )
   END_RUNG
   RUNG wire#w1
      Contact( "A0201_Profilatrice_RegolazioneFormato".AX_M[11].COut.InPosition )
      Contact( "A0201_Profilatrice_RegolazioneFormato".AX_M[12].COut.InPosition )
      S_Coil( #MB2_Decoder.OpDone )
   END_RUNG
   // the same network as SCL:
   #_w1 := #MB2_Decoder.Code = #"2284_PASSAGGIO17_COMBO_MOVE";
   "A02_HMI".MB2.Button.Profilatrice_RegolazioneFormato.Passaggio17_Combo.Bwd_Minus := #_w1 AND #MB2_Decoder.OperationMinus;
   "A02_HMI".MB2.Button.Profilatrice_RegolazioneFormato.Passaggio17_Combo.Fwd_Plus := #_w1 AND #MB2_Decoder.OperationPlus;
   IF #_w1 AND (("A0201_Profilatrice_RegolazioneFormato".AX_M[11].COut.MinusCheckNext AND "A0201_Profilatrice_RegolazioneFormato".AX_M[12].COut.MinusCheckNext) OR ("A0201_Profilatrice_RegolazioneFormato".AX_M[11].COut.PlusCheckNext AND "A0201_Profilatrice_RegolazioneFormato".AX_M[12].COut.PlusCheckNext)) THEN
       #MB2_Decoder.OpEnabled := TRUE;
   END_IF;
   IF #_w1 AND NOT "A0201_Profilatrice_RegolazioneFormato".AX_M[11].COut.Standstill AND NOT "A0201_Profilatrice_RegolazioneFormato".AX_M[12].COut.Standstill AND #MB2_Decoder.OpEnabled THEN
       #MB2_Decoder.OpRunning := TRUE;
   END_IF;
   IF #_w1 AND "A0201_Profilatrice_RegolazioneFormato".AX_M[11].COut.InPosition AND "A0201_Profilatrice_RegolazioneFormato".AX_M[12].COut.InPosition THEN
       #MB2_Decoder.OpDone := TRUE;
   END_IF;
END_REGION

REGION Network 37: MB2 Code 2285_PASSAGGIO17_COMBO_POS
   RUNG wire#powerrail
      { S7_Templates := "SrcType := Int" } EQ_Contact(in1 := #MB2_Decoder.Code, in2 := #"2285_PASSAGGIO17_COMBO_POS")
      wire#w1
      Contact( #MB2_Decoder.OperationPlus )
      Coil( "A02_HMI".MB2.Button.Profilatrice_RegolazioneFormato.Passaggio17_Combo.MoveToPos )
   END_RUNG
   RUNG wire#w1
      Contact( "A0201_Profilatrice_RegolazioneFormato".AX_M[11].COut.MinusCheckNext )
      Contact( "A0201_Profilatrice_RegolazioneFormato".AX_M[12].COut.MinusCheckNext )
      wire#w2
      S_Coil( #MB2_Decoder.OpEnabled )
   END_RUNG
   RUNG wire#w1
      Contact( "A0201_Profilatrice_RegolazioneFormato".AX_M[11].COut.PlusCheckNext )
      Contact( "A0201_Profilatrice_RegolazioneFormato".AX_M[12].COut.PlusCheckNext )
   END_RUNG wire#w2
   RUNG wire#w1
      I_Contact( "A0201_Profilatrice_RegolazioneFormato".AX_M[11].COut.Standstill )
      I_Contact( "A0201_Profilatrice_RegolazioneFormato".AX_M[12].COut.Standstill )
      Contact( #MB2_Decoder.OpEnabled )
      S_Coil( #MB2_Decoder.OpRunning )
   END_RUNG
   RUNG wire#w1
      Contact( "A0201_Profilatrice_RegolazioneFormato".AX_M[11].COut.InPosition )
      Contact( "A0201_Profilatrice_RegolazioneFormato".AX_M[12].COut.InPosition )
      S_Coil( #MB2_Decoder.OpDone )
   END_RUNG
   // the same network as SCL:
   #_w1 := #MB2_Decoder.Code = #"2285_PASSAGGIO17_COMBO_POS";
   "A02_HMI".MB2.Button.Profilatrice_RegolazioneFormato.Passaggio17_Combo.MoveToPos := #_w1 AND #MB2_Decoder.OperationPlus;
   IF #_w1 AND (("A0201_Profilatrice_RegolazioneFormato".AX_M[11].COut.MinusCheckNext AND "A0201_Profilatrice_RegolazioneFormato".AX_M[12].COut.MinusCheckNext) OR ("A0201_Profilatrice_RegolazioneFormato".AX_M[11].COut.PlusCheckNext AND "A0201_Profilatrice_RegolazioneFormato".AX_M[12].COut.PlusCheckNext)) THEN
       #MB2_Decoder.OpEnabled := TRUE;
   END_IF;
   IF #_w1 AND NOT "A0201_Profilatrice_RegolazioneFormato".AX_M[11].COut.Standstill AND NOT "A0201_Profilatrice_RegolazioneFormato".AX_M[12].COut.Standstill AND #MB2_Decoder.OpEnabled THEN
       #MB2_Decoder.OpRunning := TRUE;
   END_IF;
   IF #_w1 AND "A0201_Profilatrice_RegolazioneFormato".AX_M[11].COut.InPosition AND "A0201_Profilatrice_RegolazioneFormato".AX_M[12].COut.InPosition THEN
       #MB2_Decoder.OpDone := TRUE;
   END_IF;
END_REGION

REGION Network 38: MB2 Code 2286_PASSAGGIO18_COMBO_MOVE
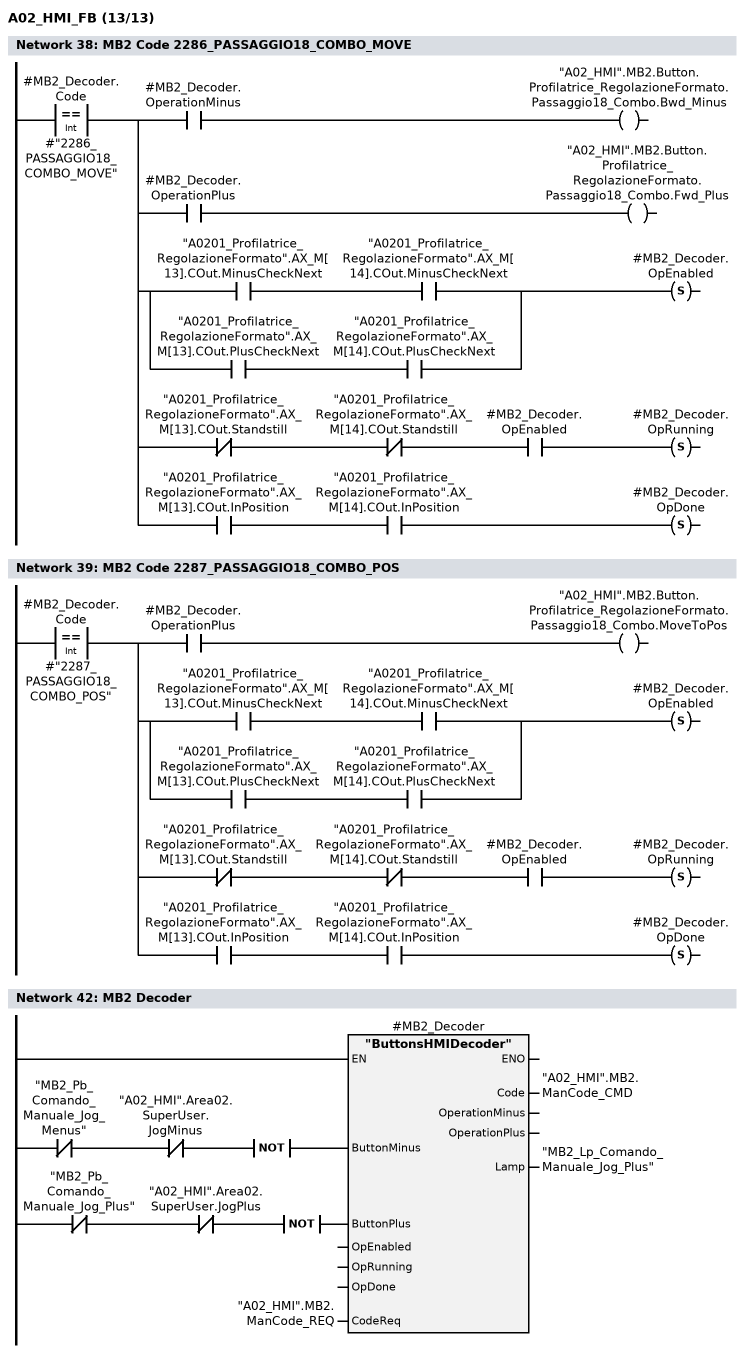
   RUNG wire#powerrail
      { S7_Templates := "SrcType := Int" } EQ_Contact(in1 := #MB2_Decoder.Code, in2 := #"2286_PASSAGGIO18_COMBO_MOVE")
      wire#w1
      Contact( #MB2_Decoder.OperationMinus )
      Coil( "A02_HMI".MB2.Button.Profilatrice_RegolazioneFormato.Passaggio18_Combo.Bwd_Minus )
   END_RUNG
   RUNG wire#w1
      Contact( #MB2_Decoder.OperationPlus )
      Coil( "A02_HMI".MB2.Button.Profilatrice_RegolazioneFormato.Passaggio18_Combo.Fwd_Plus )
   END_RUNG
   RUNG wire#w1
      Contact( "A0201_Profilatrice_RegolazioneFormato".AX_M[13].COut.MinusCheckNext )
      Contact( "A0201_Profilatrice_RegolazioneFormato".AX_M[14].COut.MinusCheckNext )
      wire#w2
      S_Coil( #MB2_Decoder.OpEnabled )
   END_RUNG
   RUNG wire#w1
      Contact( "A0201_Profilatrice_RegolazioneFormato".AX_M[13].COut.PlusCheckNext )
      Contact( "A0201_Profilatrice_RegolazioneFormato".AX_M[14].COut.PlusCheckNext )
   END_RUNG wire#w2
   RUNG wire#w1
      I_Contact( "A0201_Profilatrice_RegolazioneFormato".AX_M[13].COut.Standstill )
      I_Contact( "A0201_Profilatrice_RegolazioneFormato".AX_M[14].COut.Standstill )
      Contact( #MB2_Decoder.OpEnabled )
      S_Coil( #MB2_Decoder.OpRunning )
   END_RUNG
   RUNG wire#w1
      Contact( "A0201_Profilatrice_RegolazioneFormato".AX_M[13].COut.InPosition )
      Contact( "A0201_Profilatrice_RegolazioneFormato".AX_M[14].COut.InPosition )
      S_Coil( #MB2_Decoder.OpDone )
   END_RUNG
   // the same network as SCL:
   #_w1 := #MB2_Decoder.Code = #"2286_PASSAGGIO18_COMBO_MOVE";
   "A02_HMI".MB2.Button.Profilatrice_RegolazioneFormato.Passaggio18_Combo.Bwd_Minus := #_w1 AND #MB2_Decoder.OperationMinus;
   "A02_HMI".MB2.Button.Profilatrice_RegolazioneFormato.Passaggio18_Combo.Fwd_Plus := #_w1 AND #MB2_Decoder.OperationPlus;
   IF #_w1 AND (("A0201_Profilatrice_RegolazioneFormato".AX_M[13].COut.MinusCheckNext AND "A0201_Profilatrice_RegolazioneFormato".AX_M[14].COut.MinusCheckNext) OR ("A0201_Profilatrice_RegolazioneFormato".AX_M[13].COut.PlusCheckNext AND "A0201_Profilatrice_RegolazioneFormato".AX_M[14].COut.PlusCheckNext)) THEN
       #MB2_Decoder.OpEnabled := TRUE;
   END_IF;
   IF #_w1 AND NOT "A0201_Profilatrice_RegolazioneFormato".AX_M[13].COut.Standstill AND NOT "A0201_Profilatrice_RegolazioneFormato".AX_M[14].COut.Standstill AND #MB2_Decoder.OpEnabled THEN
       #MB2_Decoder.OpRunning := TRUE;
   END_IF;
   IF #_w1 AND "A0201_Profilatrice_RegolazioneFormato".AX_M[13].COut.InPosition AND "A0201_Profilatrice_RegolazioneFormato".AX_M[14].COut.InPosition THEN
       #MB2_Decoder.OpDone := TRUE;
   END_IF;
END_REGION

REGION Network 39: MB2 Code 2287_PASSAGGIO18_COMBO_POS
   RUNG wire#powerrail
      { S7_Templates := "SrcType := Int" } EQ_Contact(in1 := #MB2_Decoder.Code, in2 := #"2287_PASSAGGIO18_COMBO_POS")
      wire#w1
      Contact( #MB2_Decoder.OperationPlus )
      Coil( "A02_HMI".MB2.Button.Profilatrice_RegolazioneFormato.Passaggio18_Combo.MoveToPos )
   END_RUNG
   RUNG wire#w1
      Contact( "A0201_Profilatrice_RegolazioneFormato".AX_M[13].COut.MinusCheckNext )
      Contact( "A0201_Profilatrice_RegolazioneFormato".AX_M[14].COut.MinusCheckNext )
      wire#w2
      S_Coil( #MB2_Decoder.OpEnabled )
   END_RUNG
   RUNG wire#w1
      Contact( "A0201_Profilatrice_RegolazioneFormato".AX_M[13].COut.PlusCheckNext )
      Contact( "A0201_Profilatrice_RegolazioneFormato".AX_M[14].COut.PlusCheckNext )
   END_RUNG wire#w2
   RUNG wire#w1
      I_Contact( "A0201_Profilatrice_RegolazioneFormato".AX_M[13].COut.Standstill )
      I_Contact( "A0201_Profilatrice_RegolazioneFormato".AX_M[14].COut.Standstill )
      Contact( #MB2_Decoder.OpEnabled )
      S_Coil( #MB2_Decoder.OpRunning )
   END_RUNG
   RUNG wire#w1
      Contact( "A0201_Profilatrice_RegolazioneFormato".AX_M[13].COut.InPosition )
      Contact( "A0201_Profilatrice_RegolazioneFormato".AX_M[14].COut.InPosition )
      S_Coil( #MB2_Decoder.OpDone )
   END_RUNG
   // the same network as SCL:
   #_w1 := #MB2_Decoder.Code = #"2287_PASSAGGIO18_COMBO_POS";
   "A02_HMI".MB2.Button.Profilatrice_RegolazioneFormato.Passaggio18_Combo.MoveToPos := #_w1 AND #MB2_Decoder.OperationPlus;
   IF #_w1 AND (("A0201_Profilatrice_RegolazioneFormato".AX_M[13].COut.MinusCheckNext AND "A0201_Profilatrice_RegolazioneFormato".AX_M[14].COut.MinusCheckNext) OR ("A0201_Profilatrice_RegolazioneFormato".AX_M[13].COut.PlusCheckNext AND "A0201_Profilatrice_RegolazioneFormato".AX_M[14].COut.PlusCheckNext)) THEN
       #MB2_Decoder.OpEnabled := TRUE;
   END_IF;
   IF #_w1 AND NOT "A0201_Profilatrice_RegolazioneFormato".AX_M[13].COut.Standstill AND NOT "A0201_Profilatrice_RegolazioneFormato".AX_M[14].COut.Standstill AND #MB2_Decoder.OpEnabled THEN
       #MB2_Decoder.OpRunning := TRUE;
   END_IF;
   IF #_w1 AND "A0201_Profilatrice_RegolazioneFormato".AX_M[13].COut.InPosition AND "A0201_Profilatrice_RegolazioneFormato".AX_M[14].COut.InPosition THEN
       #MB2_Decoder.OpDone := TRUE;
   END_IF;
END_REGION

REGION Network 40: >
END_REGION

REGION Network 41: >
END_REGION

REGION Network 42: MB2 Decoder
   RUNG wire#powerrail
      #MB2_Decoder(ButtonMinus := wire#w1, ButtonPlus := wire#w2, OpEnabled :=, OpRunning :=, OpDone :=, CodeReq := "A02_HMI".MB2.ManCode_REQ, Code => "A02_HMI".MB2.ManCode_CMD, OperationMinus =>, OperationPlus =>, Lamp => "MB2_Lp_Comando_Manuale_Jog_Plus")
   END_RUNG
   RUNG wire#powerrail
      I_Contact( "MB2_Pb_Comando_Manuale_Jog_Menus" )
      I_Contact( "A02_HMI".Area02.SuperUser.JogMinus )
      Not()
   END_RUNG wire#w1
   RUNG wire#powerrail
      I_Contact( "MB2_Pb_Comando_Manuale_Jog_Plus" )
      I_Contact( "A02_HMI".Area02.SuperUser.JogPlus )
      Not()
   END_RUNG wire#w2
   // the same network as SCL:
   #MB2_Decoder(ButtonMinus := NOT (NOT "MB2_Pb_Comando_Manuale_Jog_Menus" AND NOT "A02_HMI".Area02.SuperUser.JogMinus),   // "ButtonsHMIDecoder"
                ButtonPlus := NOT (NOT "MB2_Pb_Comando_Manuale_Jog_Plus" AND NOT "A02_HMI".Area02.SuperUser.JogPlus),
                CodeReq := "A02_HMI".MB2.ManCode_REQ,
                Code => "A02_HMI".MB2.ManCode_CMD,
                Lamp => "MB2_Lp_Comando_Manuale_Jog_Plus");
END_REGION

REGION Network 43: >
END_REGION

REGION Network 44: >
END_REGION

REGION Network 45: >
END_REGION
END_FUNCTION_BLOCK
